METHOD FB_init : BOOL
VAR_INPUT
	bInitRetains : BOOL; // if TRUE, the retain variables are initialized (warm start / cold start)
	bInCopyCode : BOOL;  // if TRUE, the instance afterwards gets moved into the copy code (online change)
	InitialValue : ETcVnCodeDetectionModel;
END_VAR
localData := InitialValue;
AddBaseDatatype(enumBaseDatatype);
ClearReference();

AddLocalEnumeration('TCVN_CDM_DETECT_1_1', ETcVnCodeDetectionModel.TCVN_CDM_DETECT_1_1);
AddLocalEnumeration('TCVN_CDM_DETECT_1_2', ETcVnCodeDetectionModel.TCVN_CDM_DETECT_1_2);
AddLocalEnumeration('TCVN_CDM_DETECT_1_3', ETcVnCodeDetectionModel.TCVN_CDM_DETECT_1_3);
AddLocalEnumeration('TCVN_CDM_DETECT_2_1', ETcVnCodeDetectionModel.TCVN_CDM_DETECT_2_1);
AddLocalEnumeration('TCVN_CDM_DETECT_2_2', ETcVnCodeDetectionModel.TCVN_CDM_DETECT_2_2);
AddLocalEnumeration('TCVN_CDM_DETECT_2_3', ETcVnCodeDetectionModel.TCVN_CDM_DETECT_2_3);
AddLocalEnumeration('TCVN_CDM_DETECT_3_1', ETcVnCodeDetectionModel.TCVN_CDM_DETECT_3_1);
AddLocalEnumeration('TCVN_CDM_DETECT_3_2', ETcVnCodeDetectionModel.TCVN_CDM_DETECT_3_2);
AddLocalEnumeration('TCVN_CDM_DETECT_3_3', ETcVnCodeDetectionModel.TCVN_CDM_DETECT_3_3);
END_METHOD

METHOD PRIVATE AddLocalEnumeration
VAR_INPUT
	Enumeration : T_MAXSTRING;
	Value : ETcVnCodeDetectionModel;
END_VAR
AddEnumeration(Enumeration, Value);
END_METHOD

METHOD IsEnumeratorValueEqual : BOOL
VAR_INPUT
	Enumerator : I_KeyValueForwardEnumerator;
END_VAR
VAR
	storedValue : ETcVnCodeDetectionModel;
END_VAR
IF NOT Enumerator.TryGet(storedValue) THEN
	RETURN;
END_IF

IsEnumeratorValueEqual := storedValue = activeData;
END_METHOD

METHOD PUBLIC Clone : I_Datatype
VAR
    pClone : POINTER TO _ETcVnCodeDetectionModel;
END_VAR
pClone := __NEW(_ETcVnCodeDetectionModel(InitialValue := Value));
Clone := pClone^;
END_METHOD

PROPERTY PUBLIC Identifier : T_MAXSTRING
GET
Identifier := 'ETcVnCodeDetectionModel';
END_GET
END_PROPERTY

METHOD PUBLIC MakeReferenceTo
VAR_INPUT
	ReferenceTarget : REFERENCE TO ETcVnCodeDetectionModel;
END_VAR
activeData REF= ReferenceTarget;
SetBaseDatatypeReference();
END_METHOD

METHOD TryMakeReferenceTo : BOOL
VAR_INPUT
	Target : I_Datatype;
END_VAR
VAR
	pTargetData : POINTER TO ETcVnCodeDetectionModel;
END_VAR
IF NOT IsEquivalentTo(Target) THEN
	RETURN;
END_IF

pTargetData := Target.Address;
activeData REF= pTargetData^;
SetBaseDatatypeReference();
TryMakeReferenceTo := TRUE;
END_METHOD

PROPERTY PUBLIC Value : ETcVnCodeDetectionModel
GET
Value := activeData;
END_GET
SET
activeData := Value;
END_SET
END_PROPERTY

END_FUNCTION_BLOCK

// Datatypes/Enums/_ETcVnCodeType
{attribute 'linkalways'} 
{attribute 'no_explicit_call' := 'This FB is a CLASS and must be accessed using methods or properties'}
{attribute 'enable_dynamic_creation'}
FUNCTION_BLOCK _ETcVnCodeType EXTENDS EnumDatatypeBase
VAR
	localData : ETcVnCodeType;
	activeData : REFERENCE TO ETcVnCodeType;
	enumBaseDatatype : _ULINT(localData);
END_VAR

METHOD PROTECTED SetBaseDatatypeReference
VAR_INPUT
END_VAR
enumBaseDatatype.MakeReferenceTo(activeData);
END_METHOD

PROPERTY PUBLIC Address : PVOID
GET
Address := ADR(activeData);
END_GET
END_PROPERTY

METHOD PUBLIC ClearReference
VAR_INPUT
END_VAR
activeData REF= localData;
SetBaseDatatypeReference();
END_METHOD

PROPERTY PUBLIC Size : UDINT
GET
Size := SIZEOF(activeData);
END_GET
END_PROPERTY

METHOD FB_init : BOOL
VAR_INPUT
	bInitRetains : BOOL; // if TRUE, the retain variables are initialized (warm start / cold start)
	bInCopyCode : BOOL;  // if TRUE, the instance afterwards gets moved into the copy code (online change)
	InitialValue : ETcVnCodeType;
END_VAR
localData := InitialValue;
AddBaseDatatype(enumBaseDatatype);
ClearReference();

AddLocalEnumeration('TCVN_CT_ANY', ETcVnCodeType.TCVN_CT_ANY);
AddLocalEnumeration('TCVN_CT_1D', ETcVnCodeType.TCVN_CT_1D);
AddLocalEnumeration('TCVN_CT_2D', ETcVnCodeType.TCVN_CT_2D);
AddLocalEnumeration('TCVN_CT_QR', ETcVnCodeType.TCVN_CT_QR);
AddLocalEnumeration('TCVN_CT_DATAMATRIX', ETcVnCodeType.TCVN_CT_DATAMATRIX);
AddLocalEnumeration('TCVN_CT_DOTCODE', ETcVnCodeType.TCVN_CT_DOTCODE);
END_METHOD

METHOD PRIVATE AddLocalEnumeration
VAR_INPUT
	Enumeration : T_MAXSTRING;
	Value : ETcVnCodeType;
END_VAR
AddEnumeration(Enumeration, Value);
END_METHOD

METHOD IsEnumeratorValueEqual : BOOL
VAR_INPUT
	Enumerator : I_KeyValueForwardEnumerator;
END_VAR
VAR
	storedValue : ETcVnCodeType;
END_VAR
IF NOT Enumerator.TryGet(storedValue) THEN
	RETURN;
END_IF

IsEnumeratorValueEqual := storedValue = activeData;
END_METHOD

METHOD PUBLIC Clone : I_Datatype
VAR
    pClone : POINTER TO _ETcVnCodeType;
END_VAR
pClone := __NEW(_ETcVnCodeType(InitialValue := Value));
Clone := pClone^;
END_METHOD

PROPERTY PUBLIC Identifier : T_MAXSTRING
GET
Identifier := 'ETcVnCodeType';
END_GET
END_PROPERTY

METHOD PUBLIC MakeReferenceTo
VAR_INPUT
	ReferenceTarget : REFERENCE TO ETcVnCodeType;
END_VAR
activeData REF= ReferenceTarget;
SetBaseDatatypeReference();
END_METHOD

METHOD TryMakeReferenceTo : BOOL
VAR_INPUT
	Target : I_Datatype;
END_VAR
VAR
	pTargetData : POINTER TO ETcVnCodeType;
END_VAR
IF NOT IsEquivalentTo(Target) THEN
	RETURN;
END_IF

pTargetData := Target.Address;
activeData REF= pTargetData^;
SetBaseDatatypeReference();
TryMakeReferenceTo := TRUE;
END_METHOD

PROPERTY PUBLIC Value : ETcVnCodeType
GET
Value := activeData;
END_GET
SET
activeData := Value;
END_SET
END_PROPERTY

END_FUNCTION_BLOCK

// Datatypes/Enums/_ETcVnColorMap
{attribute 'linkalways'} 
{attribute 'no_explicit_call' := 'This FB is a CLASS and must be accessed using methods or properties'}
{attribute 'enable_dynamic_creation'}
FUNCTION_BLOCK _ETcVnColorMap EXTENDS EnumDatatypeBase
VAR
	localData : ETcVnColorMap;
	activeData : REFERENCE TO ETcVnColorMap;
	enumBaseDatatype : _DINT(localData);
END_VAR

METHOD PROTECTED SetBaseDatatypeReference
VAR_INPUT
END_VAR
enumBaseDatatype.MakeReferenceTo(activeData);
END_METHOD

PROPERTY PUBLIC Address : PVOID
GET
Address := ADR(activeData);
END_GET
END_PROPERTY

METHOD PUBLIC ClearReference
VAR_INPUT
END_VAR
activeData REF= localData;
SetBaseDatatypeReference();
END_METHOD

PROPERTY PUBLIC Size : UDINT
GET
Size := SIZEOF(activeData);
END_GET
END_PROPERTY

METHOD FB_init : BOOL
VAR_INPUT
	bInitRetains : BOOL; // if TRUE, the retain variables are initialized (warm start / cold start)
	bInCopyCode : BOOL;  // if TRUE, the instance afterwards gets moved into the copy code (online change)
	InitialValue : ETcVnColorMap;
END_VAR
localData := InitialValue;
AddBaseDatatype(enumBaseDatatype);
ClearReference();

AddLocalEnumeration('TCVN_CM_AUTUMN', ETcVnColorMap.TCVN_CM_AUTUMN);
AddLocalEnumeration('TCVN_CM_BONE', ETcVnColorMap.TCVN_CM_BONE);
AddLocalEnumeration('TCVN_CM_JET', ETcVnColorMap.TCVN_CM_JET);
AddLocalEnumeration('TCVN_CM_WINTER', ETcVnColorMap.TCVN_CM_WINTER);
AddLocalEnumeration('TCVN_CM_RAINBOW', ETcVnColorMap.TCVN_CM_RAINBOW);
AddLocalEnumeration('TCVN_CM_OCEAN', ETcVnColorMap.TCVN_CM_OCEAN);
AddLocalEnumeration('TCVN_CM_SUMMER', ETcVnColorMap.TCVN_CM_SUMMER);
AddLocalEnumeration('TCVN_CM_SPRING', ETcVnColorMap.TCVN_CM_SPRING);
AddLocalEnumeration('TCVN_CM_COOL', ETcVnColorMap.TCVN_CM_COOL);
AddLocalEnumeration('TCVN_CM_HSV', ETcVnColorMap.TCVN_CM_HSV);
AddLocalEnumeration('TCVN_CM_PINK', ETcVnColorMap.TCVN_CM_PINK);
AddLocalEnumeration('TCVN_CM_HOT', ETcVnColorMap.TCVN_CM_HOT);
AddLocalEnumeration('TCVN_CM_PARULA', ETcVnColorMap.TCVN_CM_PARULA);
AddLocalEnumeration('TCVN_CM_MAGMA', ETcVnColorMap.TCVN_CM_MAGMA);
AddLocalEnumeration('TCVN_CM_INFERNO', ETcVnColorMap.TCVN_CM_INFERNO);
AddLocalEnumeration('TCVN_CM_PLASMA', ETcVnColorMap.TCVN_CM_PLASMA);
AddLocalEnumeration('TCVN_CM_VIRIDIS', ETcVnColorMap.TCVN_CM_VIRIDIS);
AddLocalEnumeration('TCVN_CM_CIVIDIS', ETcVnColorMap.TCVN_CM_CIVIDIS);
AddLocalEnumeration('TCVN_CM_TWILIGHT', ETcVnColorMap.TCVN_CM_TWILIGHT);
AddLocalEnumeration('TCVN_CM_TWILIGHT_SHIFTED', ETcVnColorMap.TCVN_CM_TWILIGHT_SHIFTED);
AddLocalEnumeration('TCVN_CM_TURBO', ETcVnColorMap.TCVN_CM_TURBO);
END_METHOD

METHOD PRIVATE AddLocalEnumeration
VAR_INPUT
	Enumeration : T_MAXSTRING;
	Value : ETcVnColorMap;
END_VAR
AddEnumeration(Enumeration, Value);
END_METHOD

METHOD IsEnumeratorValueEqual : BOOL
VAR_INPUT
	Enumerator : I_KeyValueForwardEnumerator;
END_VAR
VAR
	storedValue : ETcVnColorMap;
END_VAR
IF NOT Enumerator.TryGet(storedValue) THEN
	RETURN;
END_IF

IsEnumeratorValueEqual := storedValue = activeData;
END_METHOD

METHOD PUBLIC Clone : I_Datatype
VAR
    pClone : POINTER TO _ETcVnColorMap;
END_VAR
pClone := __NEW(_ETcVnColorMap(InitialValue := Value));
Clone := pClone^;
END_METHOD

PROPERTY PUBLIC Identifier : T_MAXSTRING
GET
Identifier := 'ETcVnColorMap';
END_GET
END_PROPERTY

METHOD PUBLIC MakeReferenceTo
VAR_INPUT
	ReferenceTarget : REFERENCE TO ETcVnCalibrationPatternOrigin;
END_VAR
activeData REF= ReferenceTarget;
SetBaseDatatypeReference();
END_METHOD

METHOD TryMakeReferenceTo : BOOL
VAR_INPUT
	Target : I_Datatype;
END_VAR
VAR
	pTargetData : POINTER TO ETcVnColorMap;
END_VAR
IF NOT IsEquivalentTo(Target) THEN
	RETURN;
END_IF

pTargetData := Target.Address;
activeData REF= pTargetData^;
SetBaseDatatypeReference();
TryMakeReferenceTo := TRUE;
END_METHOD

PROPERTY PUBLIC Value : ETcVnColorMap
GET
Value := activeData;
END_GET
SET
activeData := Value;
END_SET
END_PROPERTY

END_FUNCTION_BLOCK

// Datatypes/Enums/_ETcVnColorMapSize
{attribute 'linkalways'} 
{attribute 'no_explicit_call' := 'This FB is a CLASS and must be accessed using methods or properties'}
{attribute 'enable_dynamic_creation'}
FUNCTION_BLOCK _ETcVnColorMapSize EXTENDS EnumDatatypeBase
VAR
	localData : ETcVnColorMapSize;
	activeData : REFERENCE TO ETcVnColorMapSize;
	enumBaseDatatype : _UDINT(localData);
END_VAR

METHOD PROTECTED SetBaseDatatypeReference
VAR_INPUT
END_VAR
enumBaseDatatype.MakeReferenceTo(activeData);
END_METHOD

PROPERTY PUBLIC Address : PVOID
GET
Address := ADR(activeData);
END_GET
END_PROPERTY

METHOD PUBLIC ClearReference
VAR_INPUT
END_VAR
activeData REF= localData;
SetBaseDatatypeReference();
END_METHOD

PROPERTY PUBLIC Size : UDINT
GET
Size := SIZEOF(activeData);
END_GET
END_PROPERTY

METHOD FB_init : BOOL
VAR_INPUT
	bInitRetains : BOOL; // if TRUE, the retain variables are initialized (warm start / cold start)
	bInCopyCode : BOOL;  // if TRUE, the instance afterwards gets moved into the copy code (online change)
	InitialValue : ETcVnColorMapSize;
END_VAR
localData := InitialValue;
AddBaseDatatype(enumBaseDatatype);
ClearReference();

AddLocalEnumeration('TCVN_CMS_256', ETcVnColorMapSize.TCVN_CMS_256);
AddLocalEnumeration('TCVN_CMS_65536', ETcVnColorMapSize.TCVN_CMS_65536);
END_METHOD

METHOD PRIVATE AddLocalEnumeration
VAR_INPUT
	Enumeration : T_MAXSTRING;
	Value : ETcVnColorMapSize;
END_VAR
AddEnumeration(Enumeration, Value);
END_METHOD

METHOD IsEnumeratorValueEqual : BOOL
VAR_INPUT
	Enumerator : I_KeyValueForwardEnumerator;
END_VAR
VAR
	storedValue : ETcVnColorMapSize;
END_VAR
IF NOT Enumerator.TryGet(storedValue) THEN
	RETURN;
END_IF

IsEnumeratorValueEqual := storedValue = activeData;
END_METHOD

METHOD PUBLIC Clone : I_Datatype
VAR
    pClone : POINTER TO _ETcVnColorMapSize;
END_VAR
pClone := __NEW(_ETcVnColorMapSize(InitialValue := Value));
Clone := pClone^;
END_METHOD

PROPERTY PUBLIC Identifier : T_MAXSTRING
GET
Identifier := 'ETcVnColorMapSize';
END_GET
END_PROPERTY

METHOD PUBLIC MakeReferenceTo
VAR_INPUT
	ReferenceTarget : REFERENCE TO ETcVnColorMapSize;
END_VAR
activeData REF= ReferenceTarget;
SetBaseDatatypeReference();
END_METHOD

METHOD TryMakeReferenceTo : BOOL
VAR_INPUT
	Target : I_Datatype;
END_VAR
VAR
	pTargetData : POINTER TO ETcVnColorMapSize;
END_VAR
IF NOT IsEquivalentTo(Target) THEN
	RETURN;
END_IF

pTargetData := Target.Address;
activeData REF= pTargetData^;
SetBaseDatatypeReference();
TryMakeReferenceTo := TRUE;
END_METHOD

PROPERTY PUBLIC Value : ETcVnColorMapSize
GET
Value := activeData;
END_GET
SET
activeData := Value;
END_SET
END_PROPERTY

END_FUNCTION_BLOCK

// Datatypes/Enums/_ETcVnColorSpaceTransform
{attribute 'linkalways'} 
{attribute 'no_explicit_call' := 'This FB is a CLASS and must be accessed using methods or properties'}
{attribute 'enable_dynamic_creation'}
FUNCTION_BLOCK _ETcVnColorSpaceTransform EXTENDS EnumDatatypeBase
VAR
	localData : ETcVnColorSpaceTransform;
	activeData : REFERENCE TO ETcVnColorSpaceTransform;
	enumBaseDatatype : _DINT(localData);
END_VAR

METHOD PROTECTED SetBaseDatatypeReference
VAR_INPUT
END_VAR
enumBaseDatatype.MakeReferenceTo(activeData);
END_METHOD

PROPERTY PUBLIC Address : PVOID
GET
Address := ADR(activeData);
END_GET
END_PROPERTY

METHOD PUBLIC ClearReference
VAR_INPUT
END_VAR
activeData REF= localData;
SetBaseDatatypeReference();
END_METHOD

PROPERTY PUBLIC Size : UDINT
GET
Size := SIZEOF(activeData);
END_GET
END_PROPERTY

METHOD FB_init : BOOL
VAR_INPUT
	bInitRetains : BOOL; // if TRUE, the retain variables are initialized (warm start / cold start)
	bInCopyCode : BOOL;  // if TRUE, the instance afterwards gets moved into the copy code (online change)
	InitialValue : ETcVnColorSpaceTransform;
END_VAR
localData := InitialValue;
AddBaseDatatype(enumBaseDatatype);
ClearReference();

AddLocalEnumeration('TCVN_CST_BGR_TO_BGRA', ETcVnColorSpaceTransform.TCVN_CST_BGR_TO_BGRA);
AddLocalEnumeration('TCVN_CST_RGB_TO_RGBA', ETcVnColorSpaceTransform.TCVN_CST_RGB_TO_RGBA);
AddLocalEnumeration('TCVN_CST_BGRA_TO_BGR', ETcVnColorSpaceTransform.TCVN_CST_BGRA_TO_BGR);
AddLocalEnumeration('TCVN_CST_RGBA_TO_RGB', ETcVnColorSpaceTransform.TCVN_CST_RGBA_TO_RGB);
AddLocalEnumeration('TCVN_CST_BGR_TO_RGBA', ETcVnColorSpaceTransform.TCVN_CST_BGR_TO_RGBA);
AddLocalEnumeration('TCVN_CST_RGB_TO_BGRA', ETcVnColorSpaceTransform.TCVN_CST_RGB_TO_BGRA);
AddLocalEnumeration('TCVN_CST_BGRA_TO_RGB', ETcVnColorSpaceTransform.TCVN_CST_BGRA_TO_RGB);
AddLocalEnumeration('TCVN_CST_RGBA_TO_BGR', ETcVnColorSpaceTransform.TCVN_CST_RGBA_TO_BGR);
AddLocalEnumeration('TCVN_CST_BGR_TO_RGB', ETcVnColorSpaceTransform.TCVN_CST_BGR_TO_RGB);
AddLocalEnumeration('TCVN_CST_RGB_TO_BGR', ETcVnColorSpaceTransform.TCVN_CST_RGB_TO_BGR);
AddLocalEnumeration('TCVN_CST_BGRA_TO_RGBA', ETcVnColorSpaceTransform.TCVN_CST_BGRA_TO_RGBA);
AddLocalEnumeration('TCVN_CST_RGBA_TO_BGRA', ETcVnColorSpaceTransform.TCVN_CST_RGBA_TO_BGRA);
AddLocalEnumeration('TCVN_CST_BGR_TO_GRAY', ETcVnColorSpaceTransform.TCVN_CST_BGR_TO_GRAY);
AddLocalEnumeration('TCVN_CST_RGB_TO_GRAY', ETcVnColorSpaceTransform.TCVN_CST_RGB_TO_GRAY);
AddLocalEnumeration('TCVN_CST_GRAY_TO_BGR', ETcVnColorSpaceTransform.TCVN_CST_GRAY_TO_BGR);
AddLocalEnumeration('TCVN_CST_GRAY_TO_RGB', ETcVnColorSpaceTransform.TCVN_CST_GRAY_TO_RGB);
AddLocalEnumeration('TCVN_CST_GRAY_TO_BGRA', ETcVnColorSpaceTransform.TCVN_CST_GRAY_TO_BGRA);
AddLocalEnumeration('TCVN_CST_GRAY_TO_RGBA', ETcVnColorSpaceTransform.TCVN_CST_GRAY_TO_RGBA);
AddLocalEnumeration('TCVN_CST_BGRA_TO_GRAY', ETcVnColorSpaceTransform.TCVN_CST_BGRA_TO_GRAY);
AddLocalEnumeration('TCVN_CST_RGBA_TO_GRAY', ETcVnColorSpaceTransform.TCVN_CST_RGBA_TO_GRAY);
AddLocalEnumeration('TCVN_CST_RGB_TO_BGR_565', ETcVnColorSpaceTransform.TCVN_CST_RGB_TO_BGR_565);
AddLocalEnumeration('TCVN_CST_BGR_TO_BGR_565', ETcVnColorSpaceTransform.TCVN_CST_BGR_TO_BGR_565);
AddLocalEnumeration('TCVN_CST_BGR_565_TO_RGB', ETcVnColorSpaceTransform.TCVN_CST_BGR_565_TO_RGB);
AddLocalEnumeration('TCVN_CST_BGR_565_TO_BGR', ETcVnColorSpaceTransform.TCVN_CST_BGR_565_TO_BGR);
AddLocalEnumeration('TCVN_CST_RGBA_TO_BGR_565', ETcVnColorSpaceTransform.TCVN_CST_RGBA_TO_BGR_565);
AddLocalEnumeration('TCVN_CST_BGRA_TO_BGR_565', ETcVnColorSpaceTransform.TCVN_CST_BGRA_TO_BGR_565);
AddLocalEnumeration('TCVN_CST_BGR_565_TO_RGBA', ETcVnColorSpaceTransform.TCVN_CST_BGR_565_TO_RGBA);
AddLocalEnumeration('TCVN_CST_BGR_565_TO_BGRA', ETcVnColorSpaceTransform.TCVN_CST_BGR_565_TO_BGRA);
AddLocalEnumeration('TCVN_CST_GRAY_TO_BGR_565', ETcVnColorSpaceTransform.TCVN_CST_GRAY_TO_BGR_565);
AddLocalEnumeration('TCVN_CST_BGR_565_TO_GRAY', ETcVnColorSpaceTransform.TCVN_CST_BGR_565_TO_GRAY);
AddLocalEnumeration('TCVN_CST_RGB_TO_BGR_555', ETcVnColorSpaceTransform.TCVN_CST_RGB_TO_BGR_555);
AddLocalEnumeration('TCVN_CST_BGR_TO_BGR_555', ETcVnColorSpaceTransform.TCVN_CST_BGR_TO_BGR_555);
AddLocalEnumeration('TCVN_CST_BGR_555_TO_RGB', ETcVnColorSpaceTransform.TCVN_CST_BGR_555_TO_RGB);
AddLocalEnumeration('TCVN_CST_BGR_555_TO_BGR', ETcVnColorSpaceTransform.TCVN_CST_BGR_555_TO_BGR);
AddLocalEnumeration('TCVN_CST_RGBA_TO_BGR_555', ETcVnColorSpaceTransform.TCVN_CST_RGBA_TO_BGR_555);
AddLocalEnumeration('TCVN_CST_BGRA_TO_BGR_555', ETcVnColorSpaceTransform.TCVN_CST_BGRA_TO_BGR_555);
AddLocalEnumeration('TCVN_CST_BGR_555_TO_RGBA', ETcVnColorSpaceTransform.TCVN_CST_BGR_555_TO_RGBA);
AddLocalEnumeration('TCVN_CST_BGR_555_TO_BGRA', ETcVnColorSpaceTransform.TCVN_CST_BGR_555_TO_BGRA);
AddLocalEnumeration('TCVN_CST_GRAY_TO_BGR_555', ETcVnColorSpaceTransform.TCVN_CST_GRAY_TO_BGR_555);
AddLocalEnumeration('TCVN_CST_BGR_555_TO_GRAY', ETcVnColorSpaceTransform.TCVN_CST_BGR_555_TO_GRAY);
AddLocalEnumeration('TCVN_CST_BGR_TO_XYZ', ETcVnColorSpaceTransform.TCVN_CST_BGR_TO_XYZ);
AddLocalEnumeration('TCVN_CST_RGB_TO_XYZ', ETcVnColorSpaceTransform.TCVN_CST_RGB_TO_XYZ);
AddLocalEnumeration('TCVN_CST_XYZ_TO_BGR', ETcVnColorSpaceTransform.TCVN_CST_XYZ_TO_BGR);
AddLocalEnumeration('TCVN_CST_XYZ_TO_RGB', ETcVnColorSpaceTransform.TCVN_CST_XYZ_TO_RGB);
AddLocalEnumeration('TCVN_CST_BGR_TO_YCRCB', ETcVnColorSpaceTransform.TCVN_CST_BGR_TO_YCRCB);
AddLocalEnumeration('TCVN_CST_RGB_TO_YCRCB', ETcVnColorSpaceTransform.TCVN_CST_RGB_TO_YCRCB);
AddLocalEnumeration('TCVN_CST_YCRCB_TO_BGR', ETcVnColorSpaceTransform.TCVN_CST_YCRCB_TO_BGR);
AddLocalEnumeration('TCVN_CST_YCRCB_TO_RGB', ETcVnColorSpaceTransform.TCVN_CST_YCRCB_TO_RGB);
AddLocalEnumeration('TCVN_CST_BGR_TO_HSV', ETcVnColorSpaceTransform.TCVN_CST_BGR_TO_HSV);
AddLocalEnumeration('TCVN_CST_RGB_TO_HSV', ETcVnColorSpaceTransform.TCVN_CST_RGB_TO_HSV);
AddLocalEnumeration('TCVN_CST_BGR_TO_LAB', ETcVnColorSpaceTransform.TCVN_CST_BGR_TO_LAB);
AddLocalEnumeration('TCVN_CST_RGB_TO_LAB', ETcVnColorSpaceTransform.TCVN_CST_RGB_TO_LAB);
AddLocalEnumeration('TCVN_CST_BAYER_RG_TO_BGR', ETcVnColorSpaceTransform.TCVN_CST_BAYER_RG_TO_BGR);
AddLocalEnumeration('TCVN_CST_BAYER_BG_TO_RGB', ETcVnColorSpaceTransform.TCVN_CST_BAYER_BG_TO_RGB);
AddLocalEnumeration('TCVN_CST_BAYER_GR_TO_BGR', ETcVnColorSpaceTransform.TCVN_CST_BAYER_GR_TO_BGR);
AddLocalEnumeration('TCVN_CST_BAYER_GB_TO_RGB', ETcVnColorSpaceTransform.TCVN_CST_BAYER_GB_TO_RGB);
AddLocalEnumeration('TCVN_CST_BAYER_BG_TO_BGR', ETcVnColorSpaceTransform.TCVN_CST_BAYER_BG_TO_BGR);
AddLocalEnumeration('TCVN_CST_BAYER_RG_TO_RGB', ETcVnColorSpaceTransform.TCVN_CST_BAYER_RG_TO_RGB);
AddLocalEnumeration('TCVN_CST_BAYER_GB_TO_BGR', ETcVnColorSpaceTransform.TCVN_CST_BAYER_GB_TO_BGR);
AddLocalEnumeration('TCVN_CST_BAYER_GR_TO_RGB', ETcVnColorSpaceTransform.TCVN_CST_BAYER_GR_TO_RGB);
AddLocalEnumeration('TCVN_CST_BGR_TO_LUV', ETcVnColorSpaceTransform.TCVN_CST_BGR_TO_LUV);
AddLocalEnumeration('TCVN_CST_RGB_TO_LUV', ETcVnColorSpaceTransform.TCVN_CST_RGB_TO_LUV);
AddLocalEnumeration('TCVN_CST_BGR_TO_HLS', ETcVnColorSpaceTransform.TCVN_CST_BGR_TO_HLS);
AddLocalEnumeration('TCVN_CST_RGB_TO_HLS', ETcVnColorSpaceTransform.TCVN_CST_RGB_TO_HLS);
AddLocalEnumeration('TCVN_CST_HSV_TO_BGR', ETcVnColorSpaceTransform.TCVN_CST_HSV_TO_BGR);
AddLocalEnumeration('TCVN_CST_HSV_TO_RGB', ETcVnColorSpaceTransform.TCVN_CST_HSV_TO_RGB);
AddLocalEnumeration('TCVN_CST_LAB_TO_BGR', ETcVnColorSpaceTransform.TCVN_CST_LAB_TO_BGR);
AddLocalEnumeration('TCVN_CST_LAB_TO_RGB', ETcVnColorSpaceTransform.TCVN_CST_LAB_TO_RGB);
AddLocalEnumeration('TCVN_CST_LUV_TO_BGR', ETcVnColorSpaceTransform.TCVN_CST_LUV_TO_BGR);
AddLocalEnumeration('TCVN_CST_LUV_TO_RGB', ETcVnColorSpaceTransform.TCVN_CST_LUV_TO_RGB);
AddLocalEnumeration('TCVN_CST_HLS_TO_BGR', ETcVnColorSpaceTransform.TCVN_CST_HLS_TO_BGR);
AddLocalEnumeration('TCVN_CST_HLS_TO_RGB', ETcVnColorSpaceTransform.TCVN_CST_HLS_TO_RGB);
AddLocalEnumeration('TCVN_CST_BAYER_RG_TO_BGR_VNG', ETcVnColorSpaceTransform.TCVN_CST_BAYER_RG_TO_BGR_VNG);
AddLocalEnumeration('TCVN_CST_BAYER_GR_TO_BGR_VNG', ETcVnColorSpaceTransform.TCVN_CST_BAYER_GR_TO_BGR_VNG);
AddLocalEnumeration('TCVN_CST_BAYER_BG_TO_BGR_VNG', ETcVnColorSpaceTransform.TCVN_CST_BAYER_BG_TO_BGR_VNG);
AddLocalEnumeration('TCVN_CST_BAYER_GB_TO_BGR_VNG', ETcVnColorSpaceTransform.TCVN_CST_BAYER_GB_TO_BGR_VNG);
AddLocalEnumeration('TCVN_CST_BAYER_RG_TO_RGB_VNG', ETcVnColorSpaceTransform.TCVN_CST_BAYER_RG_TO_RGB_VNG);
AddLocalEnumeration('TCVN_CST_BAYER_GR_TO_RGB_VNG', ETcVnColorSpaceTransform.TCVN_CST_BAYER_GR_TO_RGB_VNG);
AddLocalEnumeration('TCVN_CST_BAYER_BG_TO_RGB_VNG', ETcVnColorSpaceTransform.TCVN_CST_BAYER_BG_TO_RGB_VNG);
AddLocalEnumeration('TCVN_CST_BAYER_GB_TO_RGB_VNG', ETcVnColorSpaceTransform.TCVN_CST_BAYER_GB_TO_RGB_VNG);
AddLocalEnumeration('TCVN_CST_BGR_TO_HSV_FULL', ETcVnColorSpaceTransform.TCVN_CST_BGR_TO_HSV_FULL);
AddLocalEnumeration('TCVN_CST_RGB_TO_HSV_FULL', ETcVnColorSpaceTransform.TCVN_CST_RGB_TO_HSV_FULL);
AddLocalEnumeration('TCVN_CST_BGR_TO_HLS_FULL', ETcVnColorSpaceTransform.TCVN_CST_BGR_TO_HLS_FULL);
AddLocalEnumeration('TCVN_CST_RGB_TO_HLS_FULL', ETcVnColorSpaceTransform.TCVN_CST_RGB_TO_HLS_FULL);
AddLocalEnumeration('TCVN_CST_HSV_TO_BGR_FULL', ETcVnColorSpaceTransform.TCVN_CST_HSV_TO_BGR_FULL);
AddLocalEnumeration('TCVN_CST_HSV_TO_RGB_FULL', ETcVnColorSpaceTransform.TCVN_CST_HSV_TO_RGB_FULL);
AddLocalEnumeration('TCVN_CST_HLS_TO_BGR_FULL', ETcVnColorSpaceTransform.TCVN_CST_HLS_TO_BGR_FULL);
AddLocalEnumeration('TCVN_CST_HLS_TO_RGB_FULL', ETcVnColorSpaceTransform.TCVN_CST_HLS_TO_RGB_FULL);
AddLocalEnumeration('TCVN_CST_LBGR_TO_LAB', ETcVnColorSpaceTransform.TCVN_CST_LBGR_TO_LAB);
AddLocalEnumeration('TCVN_CST_LRGB_TO_LAB', ETcVnColorSpaceTransform.TCVN_CST_LRGB_TO_LAB);
AddLocalEnumeration('TCVN_CST_LBGR_TO_LUV', ETcVnColorSpaceTransform.TCVN_CST_LBGR_TO_LUV);
AddLocalEnumeration('TCVN_CST_LRGB_TO_LUV', ETcVnColorSpaceTransform.TCVN_CST_LRGB_TO_LUV);
AddLocalEnumeration('TCVN_CST_LAB_TO_LBGR', ETcVnColorSpaceTransform.TCVN_CST_LAB_TO_LBGR);
AddLocalEnumeration('TCVN_CST_LAB_TO_LRGB', ETcVnColorSpaceTransform.TCVN_CST_LAB_TO_LRGB);
AddLocalEnumeration('TCVN_CST_LUV_TO_LBGR', ETcVnColorSpaceTransform.TCVN_CST_LUV_TO_LBGR);
AddLocalEnumeration('TCVN_CST_LUV_TO_LRGB', ETcVnColorSpaceTransform.TCVN_CST_LUV_TO_LRGB);
AddLocalEnumeration('TCVN_CST_BGR_TO_YUV', ETcVnColorSpaceTransform.TCVN_CST_BGR_TO_YUV);
AddLocalEnumeration('TCVN_CST_RGB_TO_YUV', ETcVnColorSpaceTransform.TCVN_CST_RGB_TO_YUV);
AddLocalEnumeration('TCVN_CST_YUV_TO_BGR', ETcVnColorSpaceTransform.TCVN_CST_YUV_TO_BGR);
AddLocalEnumeration('TCVN_CST_YUV_TO_RGB', ETcVnColorSpaceTransform.TCVN_CST_YUV_TO_RGB);
AddLocalEnumeration('TCVN_CST_BAYER_RG_TO_GRAY', ETcVnColorSpaceTransform.TCVN_CST_BAYER_RG_TO_GRAY);
AddLocalEnumeration('TCVN_CST_BAYER_GR_TO_GRAY', ETcVnColorSpaceTransform.TCVN_CST_BAYER_GR_TO_GRAY);
AddLocalEnumeration('TCVN_CST_BAYER_BG_TO_GRAY', ETcVnColorSpaceTransform.TCVN_CST_BAYER_BG_TO_GRAY);
AddLocalEnumeration('TCVN_CST_BAYER_GB_TO_GRAY', ETcVnColorSpaceTransform.TCVN_CST_BAYER_GB_TO_GRAY);
AddLocalEnumeration('TCVN_CST_YUV_420_NV12_TO_RGB', ETcVnColorSpaceTransform.TCVN_CST_YUV_420_NV12_TO_RGB);
AddLocalEnumeration('TCVN_CST_YUV_420_NV12_TO_BGR', ETcVnColorSpaceTransform.TCVN_CST_YUV_420_NV12_TO_BGR);
AddLocalEnumeration('TCVN_CST_YUV_420_NV21_TO_RGB', ETcVnColorSpaceTransform.TCVN_CST_YUV_420_NV21_TO_RGB);
AddLocalEnumeration('TCVN_CST_YUV_420_NV21_TO_BGR', ETcVnColorSpaceTransform.TCVN_CST_YUV_420_NV21_TO_BGR);
AddLocalEnumeration('TCVN_CST_YUV_420_SP_TO_RGB', ETcVnColorSpaceTransform.TCVN_CST_YUV_420_SP_TO_RGB);
AddLocalEnumeration('TCVN_CST_YUV_420_SP_TO_BGR', ETcVnColorSpaceTransform.TCVN_CST_YUV_420_SP_TO_BGR);
AddLocalEnumeration('TCVN_CST_YUV_420_NV12_TO_RGBA', ETcVnColorSpaceTransform.TCVN_CST_YUV_420_NV12_TO_RGBA);
AddLocalEnumeration('TCVN_CST_YUV_420_NV12_TO_BGRA', ETcVnColorSpaceTransform.TCVN_CST_YUV_420_NV12_TO_BGRA);
AddLocalEnumeration('TCVN_CST_YUV_420_NV21_TO_RGBA', ETcVnColorSpaceTransform.TCVN_CST_YUV_420_NV21_TO_RGBA);
AddLocalEnumeration('TCVN_CST_YUV_420_NV21_TO_BGRA', ETcVnColorSpaceTransform.TCVN_CST_YUV_420_NV21_TO_BGRA);
AddLocalEnumeration('TCVN_CST_YUV_420_SP_TO_RGBA', ETcVnColorSpaceTransform.TCVN_CST_YUV_420_SP_TO_RGBA);
AddLocalEnumeration('TCVN_CST_YUV_420_SP_TO_BGRA', ETcVnColorSpaceTransform.TCVN_CST_YUV_420_SP_TO_BGRA);
AddLocalEnumeration('TCVN_CST_YUV_420_YV12_TO_RGB', ETcVnColorSpaceTransform.TCVN_CST_YUV_420_YV12_TO_RGB);
AddLocalEnumeration('TCVN_CST_YUV_420_YV12_TO_BGR', ETcVnColorSpaceTransform.TCVN_CST_YUV_420_YV12_TO_BGR);
AddLocalEnumeration('TCVN_CST_YUV_420_IYUV_TO_RGB', ETcVnColorSpaceTransform.TCVN_CST_YUV_420_IYUV_TO_RGB);
AddLocalEnumeration('TCVN_CST_YUV_420_IYUV_TO_BGR', ETcVnColorSpaceTransform.TCVN_CST_YUV_420_IYUV_TO_BGR);
AddLocalEnumeration('TCVN_CST_YUV_420_I420_TO_RGB', ETcVnColorSpaceTransform.TCVN_CST_YUV_420_I420_TO_RGB);
AddLocalEnumeration('TCVN_CST_YUV_420_I420_TO_BGR', ETcVnColorSpaceTransform.TCVN_CST_YUV_420_I420_TO_BGR);
AddLocalEnumeration('TCVN_CST_YUV_420_P_TO_RGB', ETcVnColorSpaceTransform.TCVN_CST_YUV_420_P_TO_RGB);
AddLocalEnumeration('TCVN_CST_YUV_420_P_TO_BGR', ETcVnColorSpaceTransform.TCVN_CST_YUV_420_P_TO_BGR);
AddLocalEnumeration('TCVN_CST_YUV_420_YV12_TO_RGBA', ETcVnColorSpaceTransform.TCVN_CST_YUV_420_YV12_TO_RGBA);
AddLocalEnumeration('TCVN_CST_YUV_420_YV12_TO_BGRA', ETcVnColorSpaceTransform.TCVN_CST_YUV_420_YV12_TO_BGRA);
AddLocalEnumeration('TCVN_CST_YUV_420_IYUV_TO_RGBA', ETcVnColorSpaceTransform.TCVN_CST_YUV_420_IYUV_TO_RGBA);
AddLocalEnumeration('TCVN_CST_YUV_420_IYUV_TO_BGRA', ETcVnColorSpaceTransform.TCVN_CST_YUV_420_IYUV_TO_BGRA);
AddLocalEnumeration('TCVN_CST_YUV_420_I420_TO_RGBA', ETcVnColorSpaceTransform.TCVN_CST_YUV_420_I420_TO_RGBA);
AddLocalEnumeration('TCVN_CST_YUV_420_I420_TO_BGRA', ETcVnColorSpaceTransform.TCVN_CST_YUV_420_I420_TO_BGRA);
AddLocalEnumeration('TCVN_CST_YUV_420_P_TO_RGBA', ETcVnColorSpaceTransform.TCVN_CST_YUV_420_P_TO_RGBA);
AddLocalEnumeration('TCVN_CST_YUV_420_P_TO_BGRA', ETcVnColorSpaceTransform.TCVN_CST_YUV_420_P_TO_BGRA);
AddLocalEnumeration('TCVN_CST_YUV_420_TO_GRAY', ETcVnColorSpaceTransform.TCVN_CST_YUV_420_TO_GRAY);
AddLocalEnumeration('TCVN_CST_YUV_420_NV21_TO_GRAY', ETcVnColorSpaceTransform.TCVN_CST_YUV_420_NV21_TO_GRAY);
AddLocalEnumeration('TCVN_CST_YUV_420_NV12_TO_GRAY', ETcVnColorSpaceTransform.TCVN_CST_YUV_420_NV12_TO_GRAY);
AddLocalEnumeration('TCVN_CST_YUV_420_YV12_TO_GRAY', ETcVnColorSpaceTransform.TCVN_CST_YUV_420_YV12_TO_GRAY);
AddLocalEnumeration('TCVN_CST_YUV_420_IYUV_TO_GRAY', ETcVnColorSpaceTransform.TCVN_CST_YUV_420_IYUV_TO_GRAY);
AddLocalEnumeration('TCVN_CST_YUV_420_I420_TO_GRAY', ETcVnColorSpaceTransform.TCVN_CST_YUV_420_I420_TO_GRAY);
AddLocalEnumeration('TCVN_CST_YUV_420_SP_TO_GRAY', ETcVnColorSpaceTransform.TCVN_CST_YUV_420_SP_TO_GRAY);
AddLocalEnumeration('TCVN_CST_YUV_420_P_TO_GRAY', ETcVnColorSpaceTransform.TCVN_CST_YUV_420_P_TO_GRAY);
AddLocalEnumeration('TCVN_CST_YUV_422_UYVY_TO_RGB', ETcVnColorSpaceTransform.TCVN_CST_YUV_422_UYVY_TO_RGB);
AddLocalEnumeration('TCVN_CST_YUV_422_UYVY_TO_BGR', ETcVnColorSpaceTransform.TCVN_CST_YUV_422_UYVY_TO_BGR);
AddLocalEnumeration('TCVN_CST_YUV_422_Y422_TO_RGB', ETcVnColorSpaceTransform.TCVN_CST_YUV_422_Y422_TO_RGB);
AddLocalEnumeration('TCVN_CST_YUV_422_Y422_TO_BGR', ETcVnColorSpaceTransform.TCVN_CST_YUV_422_Y422_TO_BGR);
AddLocalEnumeration('TCVN_CST_YUV_422_UYNV_TO_RGB', ETcVnColorSpaceTransform.TCVN_CST_YUV_422_UYNV_TO_RGB);
AddLocalEnumeration('TCVN_CST_YUV_422_UYNV_TO_BGR', ETcVnColorSpaceTransform.TCVN_CST_YUV_422_UYNV_TO_BGR);
AddLocalEnumeration('TCVN_CST_YUV_422_UYVY_TO_RGBA', ETcVnColorSpaceTransform.TCVN_CST_YUV_422_UYVY_TO_RGBA);
AddLocalEnumeration('TCVN_CST_YUV_422_UYVY_TO_BGRA', ETcVnColorSpaceTransform.TCVN_CST_YUV_422_UYVY_TO_BGRA);
AddLocalEnumeration('TCVN_CST_YUV_422_Y422_TO_RGBA', ETcVnColorSpaceTransform.TCVN_CST_YUV_422_Y422_TO_RGBA);
AddLocalEnumeration('TCVN_CST_YUV_422_Y422_TO_BGRA', ETcVnColorSpaceTransform.TCVN_CST_YUV_422_Y422_TO_BGRA);
AddLocalEnumeration('TCVN_CST_YUV_422_UYNV_TO_RGBA', ETcVnColorSpaceTransform.TCVN_CST_YUV_422_UYNV_TO_RGBA);
AddLocalEnumeration('TCVN_CST_YUV_422_UYNV_TO_BGRA', ETcVnColorSpaceTransform.TCVN_CST_YUV_422_UYNV_TO_BGRA);
AddLocalEnumeration('TCVN_CST_YUV_422_YUY2_TO_RGB', ETcVnColorSpaceTransform.TCVN_CST_YUV_422_YUY2_TO_RGB);
AddLocalEnumeration('TCVN_CST_YUV_422_YUY2_TO_BGR', ETcVnColorSpaceTransform.TCVN_CST_YUV_422_YUY2_TO_BGR);
AddLocalEnumeration('TCVN_CST_YUV_422_YVYU_TO_RGB', ETcVnColorSpaceTransform.TCVN_CST_YUV_422_YVYU_TO_RGB);
AddLocalEnumeration('TCVN_CST_YUV_422_YVYU_TO_BGR', ETcVnColorSpaceTransform.TCVN_CST_YUV_422_YVYU_TO_BGR);
AddLocalEnumeration('TCVN_CST_YUV_422_YUYV_TO_RGB', ETcVnColorSpaceTransform.TCVN_CST_YUV_422_YUYV_TO_RGB);
AddLocalEnumeration('TCVN_CST_YUV_422_YUYV_TO_BGR', ETcVnColorSpaceTransform.TCVN_CST_YUV_422_YUYV_TO_BGR);
AddLocalEnumeration('TCVN_CST_YUV_422_YUNV_TO_RGB', ETcVnColorSpaceTransform.TCVN_CST_YUV_422_YUNV_TO_RGB);
AddLocalEnumeration('TCVN_CST_YUV_422_YUNV_TO_BGR', ETcVnColorSpaceTransform.TCVN_CST_YUV_422_YUNV_TO_BGR);
AddLocalEnumeration('TCVN_CST_YUV_422_YUY2_TO_RGBA', ETcVnColorSpaceTransform.TCVN_CST_YUV_422_YUY2_TO_RGBA);
AddLocalEnumeration('TCVN_CST_YUV_422_YUY2_TO_BGRA', ETcVnColorSpaceTransform.TCVN_CST_YUV_422_YUY2_TO_BGRA);
AddLocalEnumeration('TCVN_CST_YUV_422_YVYU_TO_RGBA', ETcVnColorSpaceTransform.TCVN_CST_YUV_422_YVYU_TO_RGBA);
AddLocalEnumeration('TCVN_CST_YUV_422_YVYU_TO_BGRA', ETcVnColorSpaceTransform.TCVN_CST_YUV_422_YVYU_TO_BGRA);
AddLocalEnumeration('TCVN_CST_YUV_422_YUYV_TO_RGBA', ETcVnColorSpaceTransform.TCVN_CST_YUV_422_YUYV_TO_RGBA);
AddLocalEnumeration('TCVN_CST_YUV_422_YUYV_TO_BGRA', ETcVnColorSpaceTransform.TCVN_CST_YUV_422_YUYV_TO_BGRA);
AddLocalEnumeration('TCVN_CST_YUV_422_YUNV_TO_RGBA', ETcVnColorSpaceTransform.TCVN_CST_YUV_422_YUNV_TO_RGBA);
AddLocalEnumeration('TCVN_CST_YUV_422_YUNV_TO_BGRA', ETcVnColorSpaceTransform.TCVN_CST_YUV_422_YUNV_TO_BGRA);
AddLocalEnumeration('TCVN_CST_YUV_422_UYVY_TO_GRAY', ETcVnColorSpaceTransform.TCVN_CST_YUV_422_UYVY_TO_GRAY);
AddLocalEnumeration('TCVN_CST_YUV_422_YUY2_TO_GRAY', ETcVnColorSpaceTransform.TCVN_CST_YUV_422_YUY2_TO_GRAY);
AddLocalEnumeration('TCVN_CST_YUV_422_Y422_TO_GRAY', ETcVnColorSpaceTransform.TCVN_CST_YUV_422_Y422_TO_GRAY);
AddLocalEnumeration('TCVN_CST_YUV_422_UYNV_TO_GRAY', ETcVnColorSpaceTransform.TCVN_CST_YUV_422_UYNV_TO_GRAY);
AddLocalEnumeration('TCVN_CST_YUV_422_YVYU_TO_GRAY', ETcVnColorSpaceTransform.TCVN_CST_YUV_422_YVYU_TO_GRAY);
AddLocalEnumeration('TCVN_CST_YUV_422_YUYV_TO_GRAY', ETcVnColorSpaceTransform.TCVN_CST_YUV_422_YUYV_TO_GRAY);
AddLocalEnumeration('TCVN_CST_YUV_422_YUNV_TO_GRAY', ETcVnColorSpaceTransform.TCVN_CST_YUV_422_YUNV_TO_GRAY);
AddLocalEnumeration('TCVN_CST_RGBA_TO_PREMULTIPLICATED_RGBA', ETcVnColorSpaceTransform.TCVN_CST_RGBA_TO_PREMULTIPLICATED_RGBA);
AddLocalEnumeration('TCVN_CST_PREMULTIPLICATED_RGBA_TO_RGBA', ETcVnColorSpaceTransform.TCVN_CST_PREMULTIPLICATED_RGBA_TO_RGBA);
AddLocalEnumeration('TCVN_CST_RGB_TO_YUV_420_I420', ETcVnColorSpaceTransform.TCVN_CST_RGB_TO_YUV_420_I420);
AddLocalEnumeration('TCVN_CST_BGR_TO_YUV_420_I420', ETcVnColorSpaceTransform.TCVN_CST_BGR_TO_YUV_420_I420);
AddLocalEnumeration('TCVN_CST_RGB_TO_YUV_420_IYUV', ETcVnColorSpaceTransform.TCVN_CST_RGB_TO_YUV_420_IYUV);
AddLocalEnumeration('TCVN_CST_BGR_TO_YUV_420_IYUV', ETcVnColorSpaceTransform.TCVN_CST_BGR_TO_YUV_420_IYUV);
AddLocalEnumeration('TCVN_CST_RGBA_TO_YUV_420_I420', ETcVnColorSpaceTransform.TCVN_CST_RGBA_TO_YUV_420_I420);
AddLocalEnumeration('TCVN_CST_BGRA_TO_YUV_420_I420', ETcVnColorSpaceTransform.TCVN_CST_BGRA_TO_YUV_420_I420);
AddLocalEnumeration('TCVN_CST_RGBA_TO_YUV_420_IYUV', ETcVnColorSpaceTransform.TCVN_CST_RGBA_TO_YUV_420_IYUV);
AddLocalEnumeration('TCVN_CST_BGRA_TO_YUV_420_IYUV', ETcVnColorSpaceTransform.TCVN_CST_BGRA_TO_YUV_420_IYUV);
AddLocalEnumeration('TCVN_CST_RGB_TO_YUV_420_YV12', ETcVnColorSpaceTransform.TCVN_CST_RGB_TO_YUV_420_YV12);
AddLocalEnumeration('TCVN_CST_BGR_TO_YUV_420_YV12', ETcVnColorSpaceTransform.TCVN_CST_BGR_TO_YUV_420_YV12);
AddLocalEnumeration('TCVN_CST_RGBA_TO_YUV_420_YV12', ETcVnColorSpaceTransform.TCVN_CST_RGBA_TO_YUV_420_YV12);
AddLocalEnumeration('TCVN_CST_BGRA_TO_YUV_420_YV12', ETcVnColorSpaceTransform.TCVN_CST_BGRA_TO_YUV_420_YV12);
AddLocalEnumeration('TCVN_CST_BAYER_RG_TO_BGR_EA', ETcVnColorSpaceTransform.TCVN_CST_BAYER_RG_TO_BGR_EA);
AddLocalEnumeration('TCVN_CST_BAYER_GR_TO_BGR_EA', ETcVnColorSpaceTransform.TCVN_CST_BAYER_GR_TO_BGR_EA);
AddLocalEnumeration('TCVN_CST_BAYER_BG_TO_BGR_EA', ETcVnColorSpaceTransform.TCVN_CST_BAYER_BG_TO_BGR_EA);
AddLocalEnumeration('TCVN_CST_BAYER_GB_TO_BGR_EA', ETcVnColorSpaceTransform.TCVN_CST_BAYER_GB_TO_BGR_EA);
AddLocalEnumeration('TCVN_CST_BAYER_RG_TO_RGB_EA', ETcVnColorSpaceTransform.TCVN_CST_BAYER_RG_TO_RGB_EA);
AddLocalEnumeration('TCVN_CST_BAYER_GR_TO_RGB_EA', ETcVnColorSpaceTransform.TCVN_CST_BAYER_GR_TO_RGB_EA);
AddLocalEnumeration('TCVN_CST_BAYER_BG_TO_RGB_EA', ETcVnColorSpaceTransform.TCVN_CST_BAYER_BG_TO_RGB_EA);
AddLocalEnumeration('TCVN_CST_BAYER_GB_TO_RGB_EA', ETcVnColorSpaceTransform.TCVN_CST_BAYER_GB_TO_RGB_EA);
AddLocalEnumeration('TCVN_CST_BAYER_RG_TO_BGRA', ETcVnColorSpaceTransform.TCVN_CST_BAYER_RG_TO_BGRA);
AddLocalEnumeration('TCVN_CST_BAYER_GR_TO_BGRA', ETcVnColorSpaceTransform.TCVN_CST_BAYER_GR_TO_BGRA);
AddLocalEnumeration('TCVN_CST_BAYER_BG_TO_BGRA', ETcVnColorSpaceTransform.TCVN_CST_BAYER_BG_TO_BGRA);
AddLocalEnumeration('TCVN_CST_BAYER_GB_TO_BGRA', ETcVnColorSpaceTransform.TCVN_CST_BAYER_GB_TO_BGRA);
AddLocalEnumeration('TCVN_CST_BAYER_RG_TO_RGBA', ETcVnColorSpaceTransform.TCVN_CST_BAYER_RG_TO_RGBA);
AddLocalEnumeration('TCVN_CST_BAYER_GR_TO_RGBA', ETcVnColorSpaceTransform.TCVN_CST_BAYER_GR_TO_RGBA);
AddLocalEnumeration('TCVN_CST_BAYER_BG_TO_RGBA', ETcVnColorSpaceTransform.TCVN_CST_BAYER_BG_TO_RGBA);
AddLocalEnumeration('TCVN_CST_BAYER_GB_TO_RGBA', ETcVnColorSpaceTransform.TCVN_CST_BAYER_GB_TO_RGBA);
AddLocalEnumeration('TCVN_CST_MAX', ETcVnColorSpaceTransform.TCVN_CST_MAX);
AddLocalEnumeration('TCVN_CST_RGB_TO_YUV_422_UYVY', ETcVnColorSpaceTransform.TCVN_CST_RGB_TO_YUV_422_UYVY);
AddLocalEnumeration('TCVN_CST_BGR_TO_YUV_422_UYVY', ETcVnColorSpaceTransform.TCVN_CST_BGR_TO_YUV_422_UYVY);
AddLocalEnumeration('TCVN_CST_RGB_TO_YUV_422_Y422', ETcVnColorSpaceTransform.TCVN_CST_RGB_TO_YUV_422_Y422);
AddLocalEnumeration('TCVN_CST_BGR_TO_YUV_422_Y422', ETcVnColorSpaceTransform.TCVN_CST_BGR_TO_YUV_422_Y422);
AddLocalEnumeration('TCVN_CST_RGB_TO_YUV_422_UYNV', ETcVnColorSpaceTransform.TCVN_CST_RGB_TO_YUV_422_UYNV);
AddLocalEnumeration('TCVN_CST_BGR_TO_YUV_422_UYNV', ETcVnColorSpaceTransform.TCVN_CST_BGR_TO_YUV_422_UYNV);
AddLocalEnumeration('TCVN_CST_RGBA_TO_YUV_422_UYVY', ETcVnColorSpaceTransform.TCVN_CST_RGBA_TO_YUV_422_UYVY);
AddLocalEnumeration('TCVN_CST_BGRA_TO_YUV_422_UYVY', ETcVnColorSpaceTransform.TCVN_CST_BGRA_TO_YUV_422_UYVY);
AddLocalEnumeration('TCVN_CST_RGBA_TO_YUV_422_Y422', ETcVnColorSpaceTransform.TCVN_CST_RGBA_TO_YUV_422_Y422);
AddLocalEnumeration('TCVN_CST_BGRA_TO_YUV_422_Y422', ETcVnColorSpaceTransform.TCVN_CST_BGRA_TO_YUV_422_Y422);
AddLocalEnumeration('TCVN_CST_RGBA_TO_YUV_422_UYNV', ETcVnColorSpaceTransform.TCVN_CST_RGBA_TO_YUV_422_UYNV);
AddLocalEnumeration('TCVN_CST_BGRA_TO_YUV_422_UYNV', ETcVnColorSpaceTransform.TCVN_CST_BGRA_TO_YUV_422_UYNV);
AddLocalEnumeration('TCVN_CST_RGB_TO_YUV_422_YUY2', ETcVnColorSpaceTransform.TCVN_CST_RGB_TO_YUV_422_YUY2);
AddLocalEnumeration('TCVN_CST_BGR_TO_YUV_422_YUY2', ETcVnColorSpaceTransform.TCVN_CST_BGR_TO_YUV_422_YUY2);
AddLocalEnumeration('TCVN_CST_RGB_TO_YUV_422_YVYU', ETcVnColorSpaceTransform.TCVN_CST_RGB_TO_YUV_422_YVYU);
AddLocalEnumeration('TCVN_CST_BGR_TO_YUV_422_YVYU', ETcVnColorSpaceTransform.TCVN_CST_BGR_TO_YUV_422_YVYU);
AddLocalEnumeration('TCVN_CST_RGB_TO_YUV_422_YUYV', ETcVnColorSpaceTransform.TCVN_CST_RGB_TO_YUV_422_YUYV);
AddLocalEnumeration('TCVN_CST_BGR_TO_YUV_422_YUYV', ETcVnColorSpaceTransform.TCVN_CST_BGR_TO_YUV_422_YUYV);
AddLocalEnumeration('TCVN_CST_RGB_TO_YUV_422_YUNV', ETcVnColorSpaceTransform.TCVN_CST_RGB_TO_YUV_422_YUNV);
AddLocalEnumeration('TCVN_CST_BGR_TO_YUV_422_YUNV', ETcVnColorSpaceTransform.TCVN_CST_BGR_TO_YUV_422_YUNV);
AddLocalEnumeration('TCVN_CST_RGBA_TO_YUV_422_YUY2', ETcVnColorSpaceTransform.TCVN_CST_RGBA_TO_YUV_422_YUY2);
AddLocalEnumeration('TCVN_CST_BGRA_TO_YUV_422_YUY2', ETcVnColorSpaceTransform.TCVN_CST_BGRA_TO_YUV_422_YUY2);
AddLocalEnumeration('TCVN_CST_RGBA_TO_YUV_422_YVYU', ETcVnColorSpaceTransform.TCVN_CST_RGBA_TO_YUV_422_YVYU);
AddLocalEnumeration('TCVN_CST_BGRA_TO_YUV_422_YVYU', ETcVnColorSpaceTransform.TCVN_CST_BGRA_TO_YUV_422_YVYU);
AddLocalEnumeration('TCVN_CST_RGBA_TO_YUV_422_YUYV', ETcVnColorSpaceTransform.TCVN_CST_RGBA_TO_YUV_422_YUYV);
AddLocalEnumeration('TCVN_CST_BGRA_TO_YUV_422_YUYV', ETcVnColorSpaceTransform.TCVN_CST_BGRA_TO_YUV_422_YUYV);
AddLocalEnumeration('TCVN_CST_RGBA_TO_YUV_422_YUNV', ETcVnColorSpaceTransform.TCVN_CST_RGBA_TO_YUV_422_YUNV);
AddLocalEnumeration('TCVN_CST_BGRA_TO_YUV_422_YUNV', ETcVnColorSpaceTransform.TCVN_CST_BGRA_TO_YUV_422_YUNV);
END_METHOD

METHOD PRIVATE AddLocalEnumeration
VAR_INPUT
	Enumeration : T_MAXSTRING;
	Value : ETcVnColorSpaceTransform;
END_VAR
AddEnumeration(Enumeration, Value);
END_METHOD

METHOD IsEnumeratorValueEqual : BOOL
VAR_INPUT
	Enumerator : I_KeyValueForwardEnumerator;
END_VAR
VAR
	storedValue : ETcVnColorSpaceTransform;
END_VAR
IF NOT Enumerator.TryGet(storedValue) THEN
	RETURN;
END_IF

IsEnumeratorValueEqual := storedValue = activeData;
END_METHOD

METHOD PUBLIC Clone : I_Datatype
VAR
    pClone : POINTER TO _ETcVnColorSpaceTransform;
END_VAR
pClone := __NEW(_ETcVnColorSpaceTransform(InitialValue := Value));
Clone := pClone^;
END_METHOD

PROPERTY PUBLIC Identifier : T_MAXSTRING
GET
Identifier := 'ETcVnColorSpaceTransform';
END_GET
END_PROPERTY

METHOD PUBLIC MakeReferenceTo
VAR_INPUT
	ReferenceTarget : REFERENCE TO ETcVnColorSpaceTransform;
END_VAR
activeData REF= ReferenceTarget;
SetBaseDatatypeReference();
END_METHOD

METHOD TryMakeReferenceTo : BOOL
VAR_INPUT
	Target : I_Datatype;
END_VAR
VAR
	pTargetData : POINTER TO ETcVnColorSpaceTransform;
END_VAR
IF NOT IsEquivalentTo(Target) THEN
	RETURN;
END_IF

pTargetData := Target.Address;
activeData REF= pTargetData^;
SetBaseDatatypeReference();
TryMakeReferenceTo := TRUE;
END_METHOD

PROPERTY PUBLIC Value : ETcVnColorSpaceTransform
GET
Value := activeData;
END_GET
SET
activeData := Value;
END_SET
END_PROPERTY

END_FUNCTION_BLOCK

// Datatypes/Enums/_ETcVnColorTrainingMethod
{attribute 'linkalways'} 
{attribute 'no_explicit_call' := 'This FB is a CLASS and must be accessed using methods or properties'}
{attribute 'enable_dynamic_creation'}
FUNCTION_BLOCK _ETcVnColorTrainingMethod EXTENDS EnumDatatypeBase
VAR
	localData : ETcVnColorTrainingMethod;
	activeData : REFERENCE TO ETcVnColorTrainingMethod;
	enumBaseDatatype : _DINT(localData);
END_VAR

METHOD PROTECTED SetBaseDatatypeReference
VAR_INPUT
END_VAR
enumBaseDatatype.MakeReferenceTo(activeData);
END_METHOD

PROPERTY PUBLIC Address : PVOID
GET
Address := ADR(activeData);
END_GET
END_PROPERTY

METHOD PUBLIC ClearReference
VAR_INPUT
END_VAR
activeData REF= localData;
SetBaseDatatypeReference();
END_METHOD

PROPERTY PUBLIC Size : UDINT
GET
Size := SIZEOF(activeData);
END_GET
END_PROPERTY

METHOD FB_init : BOOL
VAR_INPUT
	bInitRetains : BOOL; // if TRUE, the retain variables are initialized (warm start / cold start)
	bInCopyCode : BOOL;  // if TRUE, the instance afterwards gets moved into the copy code (online change)
	InitialValue : ETcVnColorTrainingMethod;
END_VAR
localData := InitialValue;
AddBaseDatatype(enumBaseDatatype);
ClearReference();

AddLocalEnumeration('TCVN_CTM_LAB', ETcVnColorTrainingMethod.TCVN_CTM_LAB);
AddLocalEnumeration('TCVN_CTM_RGB', ETcVnColorTrainingMethod.TCVN_CTM_RGB);
END_METHOD

METHOD PRIVATE AddLocalEnumeration
VAR_INPUT
	Enumeration : T_MAXSTRING;
	Value : ETcVnColorTrainingMethod;
END_VAR
AddEnumeration(Enumeration, Value);
END_METHOD

METHOD IsEnumeratorValueEqual : BOOL
VAR_INPUT
	Enumerator : I_KeyValueForwardEnumerator;
END_VAR
VAR
	storedValue : ETcVnColorTrainingMethod;
END_VAR
IF NOT Enumerator.TryGet(storedValue) THEN
	RETURN;
END_IF

IsEnumeratorValueEqual := storedValue = activeData;
END_METHOD

METHOD PUBLIC Clone : I_Datatype
VAR
    pClone : POINTER TO _ETcVnColorTrainingMethod;
END_VAR
pClone := __NEW(_ETcVnColorTrainingMethod(InitialValue := Value));
Clone := pClone^;
END_METHOD

PROPERTY PUBLIC Identifier : T_MAXSTRING
GET
Identifier := 'ETcVnColorTrainingMethod';
END_GET
END_PROPERTY

METHOD PUBLIC MakeReferenceTo
VAR_INPUT
	ReferenceTarget : REFERENCE TO ETcVnColorTrainingMethod;
END_VAR
activeData REF= ReferenceTarget;
SetBaseDatatypeReference();
END_METHOD

METHOD TryMakeReferenceTo : BOOL
VAR_INPUT
	Target : I_Datatype;
END_VAR
VAR
	pTargetData : POINTER TO ETcVnColorTrainingMethod;
END_VAR
IF NOT IsEquivalentTo(Target) THEN
	RETURN;
END_IF

pTargetData := Target.Address;
activeData REF= pTargetData^;
SetBaseDatatypeReference();
TryMakeReferenceTo := TRUE;
END_METHOD

PROPERTY PUBLIC Value : ETcVnColorTrainingMethod
GET
Value := activeData;
END_GET
SET
activeData := Value;
END_SET
END_PROPERTY

END_FUNCTION_BLOCK

// Datatypes/Enums/_ETcVnComparisonOperator
{attribute 'linkalways'}
{attribute 'no_explicit_call' := 'This FB is a CLASS and must be accessed using methods or properties'}
{attribute 'enable_dynamic_creation'}
FUNCTION_BLOCK _ETcVnComparisonOperator EXTENDS EnumDatatypeBase
VAR
	localData : ETcVnComparisonOperator;
	activeData : REFERENCE TO ETcVnComparisonOperator;
	enumBaseDatatype : _INT(localData);
END_VAR

METHOD PROTECTED SetBaseDatatypeReference
VAR_INPUT
END_VAR
enumBaseDatatype.MakeReferenceTo(activeData);
END_METHOD

PROPERTY PUBLIC Address : PVOID
GET
Address := ADR(activeData);
END_GET
END_PROPERTY

METHOD PUBLIC ClearReference
VAR_INPUT
END_VAR
activeData REF= localData;
SetBaseDatatypeReference();
END_METHOD

PROPERTY PUBLIC Size : UDINT
GET
Size := SIZEOF(activeData);
END_GET
END_PROPERTY

METHOD FB_init : BOOL
VAR_INPUT
	bInitRetains : BOOL; // if TRUE, the retain variables are initialized (warm start / cold start)
	bInCopyCode : BOOL;  // if TRUE, the instance afterwards gets moved into the copy code (online change)
	InitialValue : ETcVnComparisonOperator;
END_VAR
localData := InitialValue;
AddBaseDatatype(enumBaseDatatype);
ClearReference();

AddLocalEnumeration('TCVN_CO_LESS', ETcVnComparisonOperator.TCVN_CO_LESS);
AddLocalEnumeration('TCVN_CO_GREATER', ETcVnComparisonOperator.TCVN_CO_GREATER);
END_METHOD

METHOD PRIVATE AddLocalEnumeration
VAR_INPUT
	Enumeration : T_MAXSTRING;
	Value : ETcVnComparisonOperator;
END_VAR
AddEnumeration(Enumeration, Value);
END_METHOD

METHOD IsEnumeratorValueEqual : BOOL
VAR_INPUT
	Enumerator : I_KeyValueForwardEnumerator;
END_VAR
VAR
	storedValue : ETcVnComparisonOperator;
END_VAR
IF NOT Enumerator.TryGet(storedValue) THEN
	RETURN;
END_IF

IsEnumeratorValueEqual := storedValue = activeData;
END_METHOD

METHOD PUBLIC Clone : I_Datatype
VAR
    pClone : POINTER TO _ETcVnComparisonOperator;
END_VAR
pClone := __NEW(_ETcVnComparisonOperator(InitialValue := Value));
IF pClone = 0 THEN
    RETURN;
END_IF
Clone := pClone^;
END_METHOD

PROPERTY PUBLIC Identifier : T_MAXSTRING
GET
Identifier := 'ETcVnComparisonOperator';
END_GET
END_PROPERTY

METHOD PUBLIC MakeReferenceTo
VAR_INPUT
	ReferenceTarget : REFERENCE TO ETcVnComparisonOperator;
END_VAR
activeData REF= ReferenceTarget;
SetBaseDatatypeReference();
END_METHOD

METHOD TryMakeReferenceTo : BOOL
VAR_INPUT
	Target : I_Datatype;
END_VAR
VAR
	pTargetData : POINTER TO ETcVnComparisonOperator;
END_VAR
IF NOT IsEquivalentTo(Target) THEN
	RETURN;
END_IF

pTargetData := Target.Address;
activeData REF= pTargetData^;
SetBaseDatatypeReference();
TryMakeReferenceTo := TRUE;
END_METHOD

PROPERTY PUBLIC Value : ETcVnComparisonOperator
GET
Value := activeData;
END_GET
SET
activeData := Value;
END_SET
END_PROPERTY

END_FUNCTION_BLOCK

// Datatypes/Enums/_ETcVnConnectedComponentsAlgorithm
{attribute 'linkalways'} 
{attribute 'no_explicit_call' := 'This FB is a CLASS and must be accessed using methods or properties'}
{attribute 'enable_dynamic_creation'}
FUNCTION_BLOCK _ETcVnConnectedComponentsAlgorithm EXTENDS EnumDatatypeBase
VAR
	localData : ETcVnConnectedComponentsAlgorithm;
	activeData : REFERENCE TO ETcVnConnectedComponentsAlgorithm;
	enumBaseDatatype : _DINT(localData);
END_VAR

METHOD PROTECTED SetBaseDatatypeReference
VAR_INPUT
END_VAR
enumBaseDatatype.MakeReferenceTo(activeData);
END_METHOD

PROPERTY PUBLIC Address : PVOID
GET
Address := ADR(activeData);
END_GET
END_PROPERTY

METHOD PUBLIC ClearReference
VAR_INPUT
END_VAR
activeData REF= localData;
SetBaseDatatypeReference();
END_METHOD

PROPERTY PUBLIC Size : UDINT
GET
Size := SIZEOF(activeData);
END_GET
END_PROPERTY

METHOD FB_init : BOOL
VAR_INPUT
	bInitRetains : BOOL; // if TRUE, the retain variables are initialized (warm start / cold start)
	bInCopyCode : BOOL;  // if TRUE, the instance afterwards gets moved into the copy code (online change)
	InitialValue : ETcVnConnectedComponentsAlgorithm;
END_VAR
localData := InitialValue;
AddBaseDatatype(enumBaseDatatype);
ClearReference();

AddLocalEnumeration('TCVN_CCA_WU', ETcVnConnectedComponentsAlgorithm.TCVN_CCA_WU);
AddLocalEnumeration('TCVN_CCA_GRANA', ETcVnConnectedComponentsAlgorithm.TCVN_CCA_GRANA);
END_METHOD

METHOD PRIVATE AddLocalEnumeration
VAR_INPUT
	Enumeration : T_MAXSTRING;
	Value : ETcVnConnectedComponentsAlgorithm;
END_VAR
AddEnumeration(Enumeration, Value);
END_METHOD

METHOD IsEnumeratorValueEqual : BOOL
VAR_INPUT
	Enumerator : I_KeyValueForwardEnumerator;
END_VAR
VAR
	storedValue : ETcVnConnectedComponentsAlgorithm;
END_VAR
IF NOT Enumerator.TryGet(storedValue) THEN
	RETURN;
END_IF

IsEnumeratorValueEqual := storedValue = activeData;
END_METHOD

METHOD PUBLIC Clone : I_Datatype
VAR
    pClone : POINTER TO _ETcVnConnectedComponentsAlgorithm;
END_VAR
pClone := __NEW(_ETcVnConnectedComponentsAlgorithm(InitialValue := Value));
Clone := pClone^;
END_METHOD

PROPERTY PUBLIC Identifier : T_MAXSTRING
GET
Identifier := 'ETcVnConnectedComponentsAlgorithm';
END_GET
END_PROPERTY

METHOD PUBLIC MakeReferenceTo
VAR_INPUT
	ReferenceTarget : REFERENCE TO ETcVnConnectedComponentsAlgorithm;
END_VAR
activeData REF= ReferenceTarget;
SetBaseDatatypeReference();
END_METHOD

METHOD TryMakeReferenceTo : BOOL
VAR_INPUT
	Target : I_Datatype;
END_VAR
VAR
	pTargetData : POINTER TO ETcVnConnectedComponentsAlgorithm;
END_VAR
IF NOT IsEquivalentTo(Target) THEN
	RETURN;
END_IF

pTargetData := Target.Address;
activeData REF= pTargetData^;
SetBaseDatatypeReference();
TryMakeReferenceTo := TRUE;
END_METHOD

PROPERTY PUBLIC Value : ETcVnConnectedComponentsAlgorithm
GET
Value := activeData;
END_GET
SET
activeData := Value;
END_SET
END_PROPERTY

END_FUNCTION_BLOCK

// Datatypes/Enums/_ETcVnContainerExportFormat
{attribute 'linkalways'} 
{attribute 'no_explicit_call' := 'This FB is a CLASS and must be accessed using methods or properties'}
{attribute 'enable_dynamic_creation'}
FUNCTION_BLOCK _ETcVnContainerExportFormat EXTENDS EnumDatatypeBase
VAR
	localData : ETcVnContainerExportFormat;
	activeData : REFERENCE TO ETcVnContainerExportFormat;
	enumBaseDatatype : _UINT(localData);
END_VAR

METHOD PROTECTED SetBaseDatatypeReference
VAR_INPUT
END_VAR
enumBaseDatatype.MakeReferenceTo(activeData);
END_METHOD

PROPERTY PUBLIC Address : PVOID
GET
Address := ADR(activeData);
END_GET
END_PROPERTY

METHOD PUBLIC ClearReference
VAR_INPUT
END_VAR
activeData REF= localData;
SetBaseDatatypeReference();
END_METHOD

PROPERTY PUBLIC Size : UDINT
GET
Size := SIZEOF(activeData);
END_GET
END_PROPERTY

METHOD FB_init : BOOL
VAR_INPUT
	bInitRetains : BOOL; // if TRUE, the retain variables are initialized (warm start / cold start)
	bInCopyCode : BOOL;  // if TRUE, the instance afterwards gets moved into the copy code (online change)
	InitialValue : ETcVnContainerExportFormat;
END_VAR
localData := InitialValue;
AddBaseDatatype(enumBaseDatatype);
ClearReference();

AddLocalEnumeration('TCVN_CEF_XML', ETcVnContainerExportFormat.TCVN_CEF_XML);
AddLocalEnumeration('TCVN_CEF_XML_SERIALIZED', ETcVnContainerExportFormat.TCVN_CEF_XML_SERIALIZED);
AddLocalEnumeration('TCVN_CEF_CSV', ETcVnContainerExportFormat.TCVN_CEF_CSV);
AddLocalEnumeration('TCVN_CEF_BINARY', ETcVnContainerExportFormat.TCVN_CEF_BINARY);
END_METHOD

METHOD PRIVATE AddLocalEnumeration
VAR_INPUT
	Enumeration : T_MAXSTRING;
	Value : ETcVnContainerExportFormat;
END_VAR
AddEnumeration(Enumeration, Value);
END_METHOD

METHOD IsEnumeratorValueEqual : BOOL
VAR_INPUT
	Enumerator : I_KeyValueForwardEnumerator;
END_VAR
VAR
	storedValue : ETcVnContainerExportFormat;
END_VAR
IF NOT Enumerator.TryGet(storedValue) THEN
	RETURN;
END_IF

IsEnumeratorValueEqual := storedValue = activeData;
END_METHOD

METHOD PUBLIC Clone : I_Datatype
VAR
    pClone : POINTER TO _ETcVnContainerExportFormat;
END_VAR
pClone := __NEW(_ETcVnContainerExportFormat(InitialValue := Value));
Clone := pClone^;
END_METHOD

PROPERTY PUBLIC Identifier : T_MAXSTRING
GET
Identifier := 'ETcVnContainerExportFormat';
END_GET
END_PROPERTY

METHOD PUBLIC MakeReferenceTo
VAR_INPUT
	ReferenceTarget : REFERENCE TO ETcVnContainerExportFormat;
END_VAR
activeData REF= ReferenceTarget;
SetBaseDatatypeReference();
END_METHOD

METHOD TryMakeReferenceTo : BOOL
VAR_INPUT
	Target : I_Datatype;
END_VAR
VAR
	pTargetData : POINTER TO ETcVnContainerExportFormat;
END_VAR
IF NOT IsEquivalentTo(Target) THEN
	RETURN;
END_IF

pTargetData := Target.Address;
activeData REF= pTargetData^;
SetBaseDatatypeReference();
TryMakeReferenceTo := TRUE;
END_METHOD

PROPERTY PUBLIC Value : ETcVnContainerExportFormat
GET
Value := activeData;
END_GET
SET
activeData := Value;
END_SET
END_PROPERTY

END_FUNCTION_BLOCK

// Datatypes/Enums/_ETcVnContourApproximationMethod
{attribute 'linkalways'} 
{attribute 'no_explicit_call' := 'This FB is a CLASS and must be accessed using methods or properties'}
{attribute 'enable_dynamic_creation'}
FUNCTION_BLOCK _ETcVnContourApproximationMethod EXTENDS EnumDatatypeBase
VAR
	localData : ETcVnContourApproximationMethod;
	activeData : REFERENCE TO ETcVnContourApproximationMethod;
	enumBaseDatatype : _DINT(localData);
END_VAR

METHOD PROTECTED SetBaseDatatypeReference
VAR_INPUT
END_VAR
enumBaseDatatype.MakeReferenceTo(activeData);
END_METHOD

PROPERTY PUBLIC Address : PVOID
GET
Address := ADR(activeData);
END_GET
END_PROPERTY

METHOD PUBLIC ClearReference
VAR_INPUT
END_VAR
activeData REF= localData;
SetBaseDatatypeReference();
END_METHOD

PROPERTY PUBLIC Size : UDINT
GET
Size := SIZEOF(activeData);
END_GET
END_PROPERTY

METHOD FB_init : BOOL
VAR_INPUT
	bInitRetains : BOOL; // if TRUE, the retain variables are initialized (warm start / cold start)
	bInCopyCode : BOOL;  // if TRUE, the instance afterwards gets moved into the copy code (online change)
	InitialValue : ETcVnContourApproximationMethod;
END_VAR
localData := InitialValue;
AddBaseDatatype(enumBaseDatatype);
ClearReference();

AddLocalEnumeration('TCVN_CAM_NONE', ETcVnContourApproximationMethod.TCVN_CAM_NONE);
AddLocalEnumeration('TCVN_CAM_SIMPLE', ETcVnContourApproximationMethod.TCVN_CAM_SIMPLE);
AddLocalEnumeration('TCVN_CAM_TC89_L1', ETcVnContourApproximationMethod.TCVN_CAM_TC89_L1);
AddLocalEnumeration('TCVN_CAM_TC89_KCOS', ETcVnContourApproximationMethod.TCVN_CAM_TC89_KCOS);
END_METHOD

METHOD PRIVATE AddLocalEnumeration
VAR_INPUT
	Enumeration : T_MAXSTRING;
	Value : ETcVnContourApproximationMethod;
END_VAR
AddEnumeration(Enumeration, Value);
END_METHOD

METHOD IsEnumeratorValueEqual : BOOL
VAR_INPUT
	Enumerator : I_KeyValueForwardEnumerator;
END_VAR
VAR
	storedValue : ETcVnContourApproximationMethod;
END_VAR
IF NOT Enumerator.TryGet(storedValue) THEN
	RETURN;
END_IF

IsEnumeratorValueEqual := storedValue = activeData;
END_METHOD

METHOD PUBLIC Clone : I_Datatype
VAR
    pClone : POINTER TO _ETcVnContourApproximationMethod;
END_VAR
pClone := __NEW(_ETcVnContourApproximationMethod(InitialValue := Value));
Clone := pClone^;
END_METHOD

PROPERTY PUBLIC Identifier : T_MAXSTRING
GET
Identifier := 'ETcVnContourApproximationMethod';
END_GET
END_PROPERTY

METHOD PUBLIC MakeReferenceTo
VAR_INPUT
	ReferenceTarget : REFERENCE TO ETcVnContourApproximationMethod;
END_VAR
activeData REF= ReferenceTarget;
SetBaseDatatypeReference();
END_METHOD

METHOD TryMakeReferenceTo : BOOL
VAR_INPUT
	Target : I_Datatype;
END_VAR
VAR
	pTargetData : POINTER TO ETcVnContourApproximationMethod;
END_VAR
IF NOT IsEquivalentTo(Target) THEN
	RETURN;
END_IF

pTargetData := Target.Address;
activeData REF= pTargetData^;
SetBaseDatatypeReference();
TryMakeReferenceTo := TRUE;
END_METHOD

PROPERTY PUBLIC Value : ETcVnContourApproximationMethod
GET
Value := activeData;
END_GET
SET
activeData := Value;
END_SET
END_PROPERTY

END_FUNCTION_BLOCK

// Datatypes/Enums/_ETcVnContourRetrievalMode
{attribute 'linkalways'} 
{attribute 'no_explicit_call' := 'This FB is a CLASS and must be accessed using methods or properties'}
{attribute 'enable_dynamic_creation'}
FUNCTION_BLOCK _ETcVnContourRetrievalMode EXTENDS EnumDatatypeBase
VAR
	localData : ETcVnContourRetrievalMode;
	activeData : REFERENCE TO ETcVnContourRetrievalMode;
	enumBaseDatatype : _DINT(localData);
END_VAR

METHOD PROTECTED SetBaseDatatypeReference
VAR_INPUT
END_VAR
enumBaseDatatype.MakeReferenceTo(activeData);
END_METHOD

PROPERTY PUBLIC Address : PVOID
GET
Address := ADR(activeData);
END_GET
END_PROPERTY

METHOD PUBLIC ClearReference
VAR_INPUT
END_VAR
activeData REF= localData;
SetBaseDatatypeReference();
END_METHOD

PROPERTY PUBLIC Size : UDINT
GET
Size := SIZEOF(activeData);
END_GET
END_PROPERTY

METHOD FB_init : BOOL
VAR_INPUT
	bInitRetains : BOOL; // if TRUE, the retain variables are initialized (warm start / cold start)
	bInCopyCode : BOOL;  // if TRUE, the instance afterwards gets moved into the copy code (online change)
	InitialValue : ETcVnContourRetrievalMode;
END_VAR
localData := InitialValue;
AddBaseDatatype(enumBaseDatatype);
ClearReference();

AddLocalEnumeration('TCVN_CRM_EXTERNAL', ETcVnContourRetrievalMode.TCVN_CRM_EXTERNAL);
AddLocalEnumeration('TCVN_CRM_LIST', ETcVnContourRetrievalMode.TCVN_CRM_LIST);
AddLocalEnumeration('TCVN_CRM_CONNECTED_COMPONENTS', ETcVnContourRetrievalMode.TCVN_CRM_CONNECTED_COMPONENTS);
AddLocalEnumeration('TCVN_CRM_TREE', ETcVnContourRetrievalMode.TCVN_CRM_TREE);
AddLocalEnumeration('TCVN_CRM_FLOODFILL', ETcVnContourRetrievalMode.TCVN_CRM_FLOODFILL);
END_METHOD

METHOD PRIVATE AddLocalEnumeration
VAR_INPUT
	Enumeration : T_MAXSTRING;
	Value : ETcVnContourRetrievalMode;
END_VAR
AddEnumeration(Enumeration, Value);
END_METHOD

METHOD IsEnumeratorValueEqual : BOOL
VAR_INPUT
	Enumerator : I_KeyValueForwardEnumerator;
END_VAR
VAR
	storedValue : ETcVnContourRetrievalMode;
END_VAR
IF NOT Enumerator.TryGet(storedValue) THEN
	RETURN;
END_IF

IsEnumeratorValueEqual := storedValue = activeData;
END_METHOD

METHOD PUBLIC Clone : I_Datatype
VAR
    pClone : POINTER TO _ETcVnContourRetrievalMode;
END_VAR
pClone := __NEW(_ETcVnContourRetrievalMode(InitialValue := Value));
Clone := pClone^;
END_METHOD

PROPERTY PUBLIC Identifier : T_MAXSTRING
GET
Identifier := 'ETcVnContourRetrievalMode';
END_GET
END_PROPERTY

METHOD PUBLIC MakeReferenceTo
VAR_INPUT
	ReferenceTarget : REFERENCE TO ETcVnContourRetrievalMode;
END_VAR
activeData REF= ReferenceTarget;
SetBaseDatatypeReference();
END_METHOD

METHOD TryMakeReferenceTo : BOOL
VAR_INPUT
	Target : I_Datatype;
END_VAR
VAR
	pTargetData : POINTER TO ETcVnContourRetrievalMode;
END_VAR
IF NOT IsEquivalentTo(Target) THEN
	RETURN;
END_IF

pTargetData := Target.Address;
activeData REF= pTargetData^;
SetBaseDatatypeReference();
TryMakeReferenceTo := TRUE;
END_METHOD

PROPERTY PUBLIC Value : ETcVnContourRetrievalMode
GET
Value := activeData;
END_GET
SET
activeData := Value;
END_SET
END_PROPERTY

END_FUNCTION_BLOCK

// Datatypes/Enums/_ETcVnContoursMatchComparisonMethod
{attribute 'linkalways'} 
{attribute 'no_explicit_call' := 'This FB is a CLASS and must be accessed using methods or properties'}
{attribute 'enable_dynamic_creation'}
FUNCTION_BLOCK _ETcVnContoursMatchComparisonMethod EXTENDS EnumDatatypeBase
VAR
	localData : ETcVnContoursMatchComparisonMethod;
	activeData : REFERENCE TO ETcVnContoursMatchComparisonMethod;
	enumBaseDatatype : _DINT(localData);
END_VAR

METHOD PROTECTED SetBaseDatatypeReference
VAR_INPUT
END_VAR
enumBaseDatatype.MakeReferenceTo(activeData);
END_METHOD

PROPERTY PUBLIC Address : PVOID
GET
Address := ADR(activeData);
END_GET
END_PROPERTY

METHOD PUBLIC ClearReference
VAR_INPUT
END_VAR
activeData REF= localData;
SetBaseDatatypeReference();
END_METHOD

PROPERTY PUBLIC Size : UDINT
GET
Size := SIZEOF(activeData);
END_GET
END_PROPERTY

METHOD FB_init : BOOL
VAR_INPUT
	bInitRetains : BOOL; // if TRUE, the retain variables are initialized (warm start / cold start)
	bInCopyCode : BOOL;  // if TRUE, the instance afterwards gets moved into the copy code (online change)
	InitialValue : ETcVnContoursMatchComparisonMethod;
END_VAR
localData := InitialValue;
AddBaseDatatype(enumBaseDatatype);
ClearReference();

AddLocalEnumeration('TCVN_CMCM_CONTOURS_MATCH_I1', ETcVnContoursMatchComparisonMethod.TCVN_CMCM_CONTOURS_MATCH_I1);
AddLocalEnumeration('TCVN_CMCM_CONTOURS_MATCH_I2', ETcVnContoursMatchComparisonMethod.TCVN_CMCM_CONTOURS_MATCH_I2);
AddLocalEnumeration('TCVN_CMCM_CONTOURS_MATCH_I3', ETcVnContoursMatchComparisonMethod.TCVN_CMCM_CONTOURS_MATCH_I3);
END_METHOD

METHOD PRIVATE AddLocalEnumeration
VAR_INPUT
	Enumeration : T_MAXSTRING;
	Value : ETcVnContoursMatchComparisonMethod;
END_VAR
AddEnumeration(Enumeration, Value);
END_METHOD

METHOD IsEnumeratorValueEqual : BOOL
VAR_INPUT
	Enumerator : I_KeyValueForwardEnumerator;
END_VAR
VAR
	storedValue : ETcVnContoursMatchComparisonMethod;
END_VAR
IF NOT Enumerator.TryGet(storedValue) THEN
	RETURN;
END_IF

IsEnumeratorValueEqual := storedValue = activeData;
END_METHOD

METHOD PUBLIC Clone : I_Datatype
VAR
    pClone : POINTER TO _ETcVnContoursMatchComparisonMethod;
END_VAR
pClone := __NEW(_ETcVnContoursMatchComparisonMethod(InitialValue := Value));
Clone := pClone^;
END_METHOD

PROPERTY PUBLIC Identifier : T_MAXSTRING
GET
Identifier := 'ETcVnContoursMatchComparisonMethod';
END_GET
END_PROPERTY

METHOD PUBLIC MakeReferenceTo
VAR_INPUT
	ReferenceTarget : REFERENCE TO ETcVnContoursMatchComparisonMethod;
END_VAR
activeData REF= ReferenceTarget;
SetBaseDatatypeReference();
END_METHOD

METHOD TryMakeReferenceTo : BOOL
VAR_INPUT
	Target : I_Datatype;
END_VAR
VAR
	pTargetData : POINTER TO ETcVnContoursMatchComparisonMethod;
END_VAR
IF NOT IsEquivalentTo(Target) THEN
	RETURN;
END_IF

pTargetData := Target.Address;
activeData REF= pTargetData^;
SetBaseDatatypeReference();
TryMakeReferenceTo := TRUE;
END_METHOD

PROPERTY PUBLIC Value : ETcVnContoursMatchComparisonMethod
GET
Value := activeData;
END_GET
SET
activeData := Value;
END_SET
END_PROPERTY

END_FUNCTION_BLOCK

// Datatypes/Enums/_ETcVnDataLayout
{attribute 'linkalways'} 
{attribute 'no_explicit_call' := 'This FB is a CLASS and must be accessed using methods or properties'}
{attribute 'enable_dynamic_creation'}
FUNCTION_BLOCK _ETcVnDataLayout EXTENDS EnumDatatypeBase
VAR
	localData : ETcVnDataLayout;
	activeData : REFERENCE TO ETcVnDataLayout;
	enumBaseDatatype : _ULINT(localData);
END_VAR

METHOD PROTECTED SetBaseDatatypeReference
VAR_INPUT
END_VAR
enumBaseDatatype.MakeReferenceTo(activeData);
END_METHOD

PROPERTY PUBLIC Address : PVOID
GET
Address := ADR(activeData);
END_GET
END_PROPERTY

METHOD PUBLIC ClearReference
VAR_INPUT
END_VAR
activeData REF= localData;
SetBaseDatatypeReference();
END_METHOD

PROPERTY PUBLIC Size : UDINT
GET
Size := SIZEOF(activeData);
END_GET
END_PROPERTY

METHOD FB_init : BOOL
VAR_INPUT
	bInitRetains : BOOL; // if TRUE, the retain variables are initialized (warm start / cold start)
	bInCopyCode : BOOL;  // if TRUE, the instance afterwards gets moved into the copy code (online change)
	InitialValue : ETcVnDataLayout;
END_VAR
localData := InitialValue;
AddBaseDatatype(enumBaseDatatype);
ClearReference();

AddLocalEnumeration('TCVN_DL_DEFAULT', ETcVnDataLayout.TCVN_DL_DEFAULT);
AddLocalEnumeration('TCVN_DL_2D_HW', ETcVnDataLayout.TCVN_DL_2D_HW);
AddLocalEnumeration('TCVN_DL_2D_WH', ETcVnDataLayout.TCVN_DL_2D_WH);
AddLocalEnumeration('TCVN_DL_3D_CHW', ETcVnDataLayout.TCVN_DL_3D_CHW);
AddLocalEnumeration('TCVN_DL_3D_HWC', ETcVnDataLayout.TCVN_DL_3D_HWC);
AddLocalEnumeration('TCVN_DL_4D_NCHW', ETcVnDataLayout.TCVN_DL_4D_NCHW);
AddLocalEnumeration('TCVN_DL_4D_NHWC', ETcVnDataLayout.TCVN_DL_4D_NHWC);
END_METHOD

METHOD PRIVATE AddLocalEnumeration
VAR_INPUT
	Enumeration : T_MAXSTRING;
	Value : ETcVnDataLayout;
END_VAR
AddEnumeration(Enumeration, Value);
END_METHOD

METHOD IsEnumeratorValueEqual : BOOL
VAR_INPUT
	Enumerator : I_KeyValueForwardEnumerator;
END_VAR
VAR
	storedValue : ETcVnDataLayout;
END_VAR
IF NOT Enumerator.TryGet(storedValue) THEN
	RETURN;
END_IF

IsEnumeratorValueEqual := storedValue = activeData;
END_METHOD

METHOD PUBLIC Clone : I_Datatype
VAR
    pClone : POINTER TO _ETcVnDataLayout;
END_VAR
pClone := __NEW(_ETcVnDataLayout(InitialValue := Value));
Clone := pClone^;
END_METHOD

PROPERTY PUBLIC Identifier : T_MAXSTRING
GET
Identifier := 'ETcVnDataLayout';
END_GET
END_PROPERTY

METHOD PUBLIC MakeReferenceTo
VAR_INPUT
	ReferenceTarget : REFERENCE TO ETcVnDataLayout;
END_VAR
activeData REF= ReferenceTarget;
SetBaseDatatypeReference();
END_METHOD

METHOD TryMakeReferenceTo : BOOL
VAR_INPUT
	Target : I_Datatype;
END_VAR
VAR
	pTargetData : POINTER TO ETcVnDataLayout;
END_VAR
IF NOT IsEquivalentTo(Target) THEN
	RETURN;
END_IF

pTargetData := Target.Address;
activeData REF= pTargetData^;
SetBaseDatatypeReference();
TryMakeReferenceTo := TRUE;
END_METHOD

PROPERTY PUBLIC Value : ETcVnDataLayout
GET
Value := activeData;
END_GET
SET
activeData := Value;
END_SET
END_PROPERTY

END_FUNCTION_BLOCK

// Datatypes/Enums/_ETcVnDataMatrixOptions
{attribute 'linkalways'} 
{attribute 'no_explicit_call' := 'This FB is a CLASS and must be accessed using methods or properties'}
{attribute 'enable_dynamic_creation'}
FUNCTION_BLOCK _ETcVnDataMatrixOptions EXTENDS EnumDatatypeBase
VAR
	localData : ETcVnDataMatrixOptions;
	activeData : REFERENCE TO ETcVnDataMatrixOptions;
	enumBaseDatatype : _ULINT(localData);
END_VAR

METHOD PROTECTED SetBaseDatatypeReference
VAR_INPUT
END_VAR
enumBaseDatatype.MakeReferenceTo(activeData);
END_METHOD

PROPERTY PUBLIC Address : PVOID
GET
Address := ADR(activeData);
END_GET
END_PROPERTY

METHOD PUBLIC ClearReference
VAR_INPUT
END_VAR
activeData REF= localData;
SetBaseDatatypeReference();
END_METHOD

PROPERTY PUBLIC Size : UDINT
GET
Size := SIZEOF(activeData);
END_GET
END_PROPERTY

METHOD FB_init : BOOL
VAR_INPUT
	bInitRetains : BOOL; // if TRUE, the retain variables are initialized (warm start / cold start)
	bInCopyCode : BOOL;  // if TRUE, the instance afterwards gets moved into the copy code (online change)
	InitialValue : ETcVnDataMatrixOptions;
END_VAR
localData := InitialValue;
AddBaseDatatype(enumBaseDatatype);
ClearReference();

AddLocalEnumeration('TCVN_DMO_DEFAULT', ETcVnDataMatrixOptions.TCVN_DMO_DEFAULT);
AddLocalEnumeration('TCVN_DMO_BINARY_INPUT', ETcVnDataMatrixOptions.TCVN_DMO_BINARY_INPUT);
AddLocalEnumeration('TCVN_DMO_GLOBAL_THRESHOLD', ETcVnDataMatrixOptions.TCVN_DMO_GLOBAL_THRESHOLD);
AddLocalEnumeration('TCVN_DMO_BINARY_GRID', ETcVnDataMatrixOptions.TCVN_DMO_BINARY_GRID);
AddLocalEnumeration('TCVN_DMO_STATIC_GRID', ETcVnDataMatrixOptions.TCVN_DMO_STATIC_GRID);
AddLocalEnumeration('TCVN_DMO_REGULAR_COLOR', ETcVnDataMatrixOptions.TCVN_DMO_REGULAR_COLOR);
AddLocalEnumeration('TCVN_DMO_INVERTED_COLOR', ETcVnDataMatrixOptions.TCVN_DMO_INVERTED_COLOR);
END_METHOD

METHOD PRIVATE AddLocalEnumeration
VAR_INPUT
	Enumeration : T_MAXSTRING;
	Value : ETcVnDataMatrixOptions;
END_VAR
AddEnumeration(Enumeration, Value);
END_METHOD

METHOD IsEnumeratorValueEqual : BOOL
VAR_INPUT
	Enumerator : I_KeyValueForwardEnumerator;
END_VAR
VAR
	storedValue : ETcVnDataMatrixOptions;
END_VAR
IF NOT Enumerator.TryGet(storedValue) THEN
	RETURN;
END_IF

IsEnumeratorValueEqual := storedValue = activeData;
END_METHOD

METHOD PUBLIC Clone : I_Datatype
VAR
    pClone : POINTER TO _ETcVnDataMatrixOptions;
END_VAR
pClone := __NEW(_ETcVnDataMatrixOptions(InitialValue := Value));
Clone := pClone^;
END_METHOD

PROPERTY PUBLIC Identifier : T_MAXSTRING
GET
Identifier := 'ETcVnDataMatrixOptions';
END_GET
END_PROPERTY

METHOD PUBLIC MakeReferenceTo
VAR_INPUT
	ReferenceTarget : REFERENCE TO ETcVnDataMatrixOptions;
END_VAR
activeData REF= ReferenceTarget;
SetBaseDatatypeReference();
END_METHOD

METHOD TryMakeReferenceTo : BOOL
VAR_INPUT
	Target : I_Datatype;
END_VAR
VAR
	pTargetData : POINTER TO ETcVnDataMatrixOptions;
END_VAR
IF NOT IsEquivalentTo(Target) THEN
	RETURN;
END_IF

pTargetData := Target.Address;
activeData REF= pTargetData^;
SetBaseDatatypeReference();
TryMakeReferenceTo := TRUE;
END_METHOD

PROPERTY PUBLIC Value : ETcVnDataMatrixOptions
GET
Value := activeData;
END_GET
SET
activeData := Value;
END_SET
END_PROPERTY

END_FUNCTION_BLOCK

// Datatypes/Enums/_ETcVnDetectBarcodesWalshOptions
{attribute 'linkalways'}
{attribute 'no_explicit_call' := 'This FB is a CLASS and must be accessed using methods or properties'}
{attribute 'enable_dynamic_creation'}
FUNCTION_BLOCK _ETcVnDetectBarcodesWalshOptions EXTENDS EnumDatatypeBase
VAR
	localData : ETcVnDetectBarcodesWalshOptions;
	activeData : REFERENCE TO ETcVnDetectBarcodesWalshOptions;
	enumBaseDatatype : _UDINT(localData);
END_VAR

METHOD PROTECTED SetBaseDatatypeReference
VAR_INPUT
END_VAR
enumBaseDatatype.MakeReferenceTo(activeData);
END_METHOD

PROPERTY PUBLIC Address : PVOID
GET
Address := ADR(activeData);
END_GET
END_PROPERTY

METHOD PUBLIC ClearReference
VAR_INPUT
END_VAR
activeData REF= localData;
SetBaseDatatypeReference();
END_METHOD

PROPERTY PUBLIC Size : UDINT
GET
Size := SIZEOF(activeData);
END_GET
END_PROPERTY

METHOD FB_init : BOOL
VAR_INPUT
	bInitRetains : BOOL; // if TRUE, the retain variables are initialized (warm start / cold start)
	bInCopyCode : BOOL;  // if TRUE, the instance afterwards gets moved into the copy code (online change)
	InitialValue : ETcVnDetectBarcodesWalshOptions;
END_VAR
localData := InitialValue;
AddBaseDatatype(enumBaseDatatype);
ClearReference();

AddLocalEnumeration('TCVN_DBWO_HORIZONTAL', ETcVnDetectBarcodesWalshOptions.TCVN_DBWO_HORIZONTAL);
AddLocalEnumeration('TCVN_DBWO_VERTICAL', ETcVnDetectBarcodesWalshOptions.TCVN_DBWO_VERTICAL);
AddLocalEnumeration('TCVN_DBWO_DIAGONAL_45', ETcVnDetectBarcodesWalshOptions.TCVN_DBWO_DIAGONAL_45);
AddLocalEnumeration('TCVN_DBWO_DIAGONAL_135', ETcVnDetectBarcodesWalshOptions.TCVN_DBWO_DIAGONAL_135);
AddLocalEnumeration('TCVN_DBWO_ALL_DIRECTIONS', ETcVnDetectBarcodesWalshOptions.TCVN_DBWO_ALL_DIRECTIONS);
END_METHOD

METHOD PRIVATE AddLocalEnumeration
VAR_INPUT
	Enumeration : T_MAXSTRING;
	Value : ETcVnDetectBarcodesWalshOptions;
END_VAR
AddEnumeration(Enumeration, Value);
END_METHOD

METHOD IsEnumeratorValueEqual : BOOL
VAR_INPUT
	Enumerator : I_KeyValueForwardEnumerator;
END_VAR
VAR
	storedValue : ETcVnDetectBarcodesWalshOptions;
END_VAR
IF NOT Enumerator.TryGet(storedValue) THEN
	RETURN;
END_IF

IsEnumeratorValueEqual := storedValue = activeData;
END_METHOD

METHOD PUBLIC Clone : I_Datatype
VAR
    pClone : POINTER TO _ETcVnDetectBarcodesWalshOptions;
END_VAR
pClone := __NEW(_ETcVnDetectBarcodesWalshOptions(InitialValue := Value));
IF pClone = 0 THEN
    RETURN;
END_IF
Clone := pClone^;
END_METHOD

PROPERTY PUBLIC Identifier : T_MAXSTRING
GET
Identifier := 'ETcVnDetectBarcodesWalshOptions';
END_GET
END_PROPERTY

METHOD PUBLIC MakeReferenceTo
VAR_INPUT
	ReferenceTarget : REFERENCE TO ETcVnDetectBarcodesWalshOptions;
END_VAR
activeData REF= ReferenceTarget;
SetBaseDatatypeReference();
END_METHOD

METHOD TryMakeReferenceTo : BOOL
VAR_INPUT
	Target : I_Datatype;
END_VAR
VAR
	pTargetData : POINTER TO ETcVnDetectBarcodesWalshOptions;
END_VAR
IF NOT IsEquivalentTo(Target) THEN
	RETURN;
END_IF

pTargetData := Target.Address;
activeData REF= pTargetData^;
SetBaseDatatypeReference();
TryMakeReferenceTo := TRUE;
END_METHOD

PROPERTY PUBLIC Value : ETcVnDetectBarcodesWalshOptions
GET
Value := activeData;
END_GET
SET
activeData := Value;
END_SET
END_PROPERTY

END_FUNCTION_BLOCK

// Datatypes/Enums/_ETcVnDetectPatternPointsOptions
{attribute 'linkalways'}
{attribute 'no_explicit_call' := 'This FB is a CLASS and must be accessed using methods or properties'}
{attribute 'enable_dynamic_creation'}
FUNCTION_BLOCK _ETcVnDetectPatternPointsOptions EXTENDS EnumDatatypeBase
VAR
	localData : ETcVnDetectPatternPointsOptions;
	activeData : REFERENCE TO ETcVnDetectPatternPointsOptions;
	enumBaseDatatype : _UDINT(localData);
END_VAR

METHOD PROTECTED SetBaseDatatypeReference
VAR_INPUT
END_VAR
enumBaseDatatype.MakeReferenceTo(activeData);
END_METHOD

PROPERTY PUBLIC Address : PVOID
GET
Address := ADR(activeData);
END_GET
END_PROPERTY

METHOD PUBLIC ClearReference
VAR_INPUT
END_VAR
activeData REF= localData;
SetBaseDatatypeReference();
END_METHOD

PROPERTY PUBLIC Size : UDINT
GET
Size := SIZEOF(activeData);
END_GET
END_PROPERTY

METHOD FB_init : BOOL
VAR_INPUT
	bInitRetains : BOOL; // if TRUE, the retain variables are initialized (warm start / cold start)
	bInCopyCode : BOOL;  // if TRUE, the instance afterwards gets moved into the copy code (online change)
	InitialValue : ETcVnDetectPatternPointsOptions;
END_VAR
localData := InitialValue;
AddBaseDatatype(enumBaseDatatype);
ClearReference();

AddLocalEnumeration('TCVN_DPPO_SYMMETRIC', ETcVnDetectPatternPointsOptions.TCVN_DPPO_SYMMETRIC);
AddLocalEnumeration('TCVN_DPPO_ASYMMETRIC', ETcVnDetectPatternPointsOptions.TCVN_DPPO_ASYMMETRIC);
AddLocalEnumeration('TCVN_DPPO_CLUSTERING', ETcVnDetectPatternPointsOptions.TCVN_DPPO_CLUSTERING);
END_METHOD

METHOD PRIVATE AddLocalEnumeration
VAR_INPUT
	Enumeration : T_MAXSTRING;
	Value : ETcVnDetectPatternPointsOptions;
END_VAR
AddEnumeration(Enumeration, Value);
END_METHOD

METHOD IsEnumeratorValueEqual : BOOL
VAR_INPUT
	Enumerator : I_KeyValueForwardEnumerator;
END_VAR
VAR
	storedValue : ETcVnDetectPatternPointsOptions;
END_VAR
IF NOT Enumerator.TryGet(storedValue) THEN
	RETURN;
END_IF

IsEnumeratorValueEqual := storedValue = activeData;
END_METHOD

METHOD PUBLIC Clone : I_Datatype
VAR
    pClone : POINTER TO _ETcVnDetectPatternPointsOptions;
END_VAR
pClone := __NEW(_ETcVnDetectPatternPointsOptions(InitialValue := Value));
IF pClone = 0 THEN
    RETURN;
END_IF
Clone := pClone^;
END_METHOD

PROPERTY PUBLIC Identifier : T_MAXSTRING
GET
Identifier := 'ETcVnDetectPatternPointsOptions';
END_GET
END_PROPERTY

METHOD PUBLIC MakeReferenceTo
VAR_INPUT
	ReferenceTarget : REFERENCE TO ETcVnDetectPatternPointsOptions;
END_VAR
activeData REF= ReferenceTarget;
SetBaseDatatypeReference();
END_METHOD

METHOD TryMakeReferenceTo : BOOL
VAR_INPUT
	Target : I_Datatype;
END_VAR
VAR
	pTargetData : POINTER TO ETcVnDetectPatternPointsOptions;
END_VAR
IF NOT IsEquivalentTo(Target) THEN
	RETURN;
END_IF

pTargetData := Target.Address;
activeData REF= pTargetData^;
SetBaseDatatypeReference();
TryMakeReferenceTo := TRUE;
END_METHOD

PROPERTY PUBLIC Value : ETcVnDetectPatternPointsOptions
GET
Value := activeData;
END_GET
SET
activeData := Value;
END_SET
END_PROPERTY

END_FUNCTION_BLOCK

// Datatypes/Enums/_ETcVnDiffusivityTypeKAZE
{attribute 'linkalways'} 
{attribute 'no_explicit_call' := 'This FB is a CLASS and must be accessed using methods or properties'}
{attribute 'enable_dynamic_creation'}
FUNCTION_BLOCK _ETcVnDiffusivityTypeKAZE EXTENDS EnumDatatypeBase
VAR
	localData : ETcVnDiffusivityTypeKAZE;
	activeData : REFERENCE TO ETcVnDiffusivityTypeKAZE;
	enumBaseDatatype : _DINT(localData);
END_VAR

METHOD PROTECTED SetBaseDatatypeReference
VAR_INPUT
END_VAR
enumBaseDatatype.MakeReferenceTo(activeData);
END_METHOD

PROPERTY PUBLIC Address : PVOID
GET
Address := ADR(activeData);
END_GET
END_PROPERTY

METHOD PUBLIC ClearReference
VAR_INPUT
END_VAR
activeData REF= localData;
SetBaseDatatypeReference();
END_METHOD

PROPERTY PUBLIC Size : UDINT
GET
Size := SIZEOF(activeData);
END_GET
END_PROPERTY

METHOD FB_init : BOOL
VAR_INPUT
	bInitRetains : BOOL; // if TRUE, the retain variables are initialized (warm start / cold start)
	bInCopyCode : BOOL;  // if TRUE, the instance afterwards gets moved into the copy code (online change)
	InitialValue : ETcVnDiffusivityTypeKAZE;
END_VAR
localData := InitialValue;
AddBaseDatatype(enumBaseDatatype);
ClearReference();

AddLocalEnumeration('TCVN_DT1_KAZE_PM_G1', ETcVnDiffusivityTypeKAZE.TCVN_DT1_KAZE_PM_G1);
AddLocalEnumeration('TCVN_DT1_KAZE_PM_G2', ETcVnDiffusivityTypeKAZE.TCVN_DT1_KAZE_PM_G2);
AddLocalEnumeration('TCVN_DT1_KAZE_WEICKERT', ETcVnDiffusivityTypeKAZE.TCVN_DT1_KAZE_WEICKERT);
AddLocalEnumeration('TCVN_DT1_KAZE_CHARBONNIER', ETcVnDiffusivityTypeKAZE.TCVN_DT1_KAZE_CHARBONNIER);
END_METHOD

METHOD PRIVATE AddLocalEnumeration
VAR_INPUT
	Enumeration : T_MAXSTRING;
	Value : ETcVnDiffusivityTypeKAZE;
END_VAR
AddEnumeration(Enumeration, Value);
END_METHOD

METHOD IsEnumeratorValueEqual : BOOL
VAR_INPUT
	Enumerator : I_KeyValueForwardEnumerator;
END_VAR
VAR
	storedValue : ETcVnDiffusivityTypeKAZE;
END_VAR
IF NOT Enumerator.TryGet(storedValue) THEN
	RETURN;
END_IF

IsEnumeratorValueEqual := storedValue = activeData;
END_METHOD

METHOD PUBLIC Clone : I_Datatype
VAR
    pClone : POINTER TO _ETcVnDiffusivityTypeKAZE;
END_VAR
pClone := __NEW(_ETcVnDiffusivityTypeKAZE(InitialValue := Value));
Clone := pClone^;
END_METHOD

PROPERTY PUBLIC Identifier : T_MAXSTRING
GET
Identifier := 'ETcVnDiffusivityTypeKAZE';
END_GET
END_PROPERTY

METHOD PUBLIC MakeReferenceTo
VAR_INPUT
	ReferenceTarget : REFERENCE TO ETcVnDiffusivityTypeKAZE;
END_VAR
activeData REF= ReferenceTarget;
SetBaseDatatypeReference();
END_METHOD

METHOD TryMakeReferenceTo : BOOL
VAR_INPUT
	Target : I_Datatype;
END_VAR
VAR
	pTargetData : POINTER TO ETcVnDiffusivityTypeKAZE;
END_VAR
IF NOT IsEquivalentTo(Target) THEN
	RETURN;
END_IF

pTargetData := Target.Address;
activeData REF= pTargetData^;
SetBaseDatatypeReference();
TryMakeReferenceTo := TRUE;
END_METHOD

PROPERTY PUBLIC Value : ETcVnDiffusivityTypeKAZE
GET
Value := activeData;
END_GET
SET
activeData := Value;
END_SET
END_PROPERTY

END_FUNCTION_BLOCK

// Datatypes/Enums/_ETcVnDistanceTransformationLabel
{attribute 'linkalways'} 
{attribute 'no_explicit_call' := 'This FB is a CLASS and must be accessed using methods or properties'}
{attribute 'enable_dynamic_creation'}
FUNCTION_BLOCK _ETcVnDistanceTransformationLabel EXTENDS EnumDatatypeBase
VAR
	localData : ETcVnDistanceTransformationLabel;
	activeData : REFERENCE TO ETcVnDistanceTransformationLabel;
	enumBaseDatatype : _DINT(localData);
END_VAR

METHOD PROTECTED SetBaseDatatypeReference
VAR_INPUT
END_VAR
enumBaseDatatype.MakeReferenceTo(activeData);
END_METHOD

PROPERTY PUBLIC Address : PVOID
GET
Address := ADR(activeData);
END_GET
END_PROPERTY

METHOD PUBLIC ClearReference
VAR_INPUT
END_VAR
activeData REF= localData;
SetBaseDatatypeReference();
END_METHOD

PROPERTY PUBLIC Size : UDINT
GET
Size := SIZEOF(activeData);
END_GET
END_PROPERTY

METHOD FB_init : BOOL
VAR_INPUT
	bInitRetains : BOOL; // if TRUE, the retain variables are initialized (warm start / cold start)
	bInCopyCode : BOOL;  // if TRUE, the instance afterwards gets moved into the copy code (online change)
	InitialValue : ETcVnDistanceTransformationLabel;
END_VAR
localData := InitialValue;
AddBaseDatatype(enumBaseDatatype);
ClearReference();

AddLocalEnumeration('TCVN_DTL_CCOMP', ETcVnDistanceTransformationLabel.TCVN_DTL_CCOMP);
AddLocalEnumeration('TCVN_DTL_PIXEL', ETcVnDistanceTransformationLabel.TCVN_DTL_PIXEL);
END_METHOD

METHOD PRIVATE AddLocalEnumeration
VAR_INPUT
	Enumeration : T_MAXSTRING;
	Value : ETcVnDistanceTransformationLabel;
END_VAR
AddEnumeration(Enumeration, Value);
END_METHOD

METHOD IsEnumeratorValueEqual : BOOL
VAR_INPUT
	Enumerator : I_KeyValueForwardEnumerator;
END_VAR
VAR
	storedValue : ETcVnDistanceTransformationLabel;
END_VAR
IF NOT Enumerator.TryGet(storedValue) THEN
	RETURN;
END_IF

IsEnumeratorValueEqual := storedValue = activeData;
END_METHOD

METHOD PUBLIC Clone : I_Datatype
VAR
    pClone : POINTER TO _ETcVnDistanceTransformationLabel;
END_VAR
pClone := __NEW(_ETcVnDistanceTransformationLabel(InitialValue := Value));
Clone := pClone^;
END_METHOD

PROPERTY PUBLIC Identifier : T_MAXSTRING
GET
Identifier := 'ETcVnDistanceTransformationLabel';
END_GET
END_PROPERTY

METHOD PUBLIC MakeReferenceTo
VAR_INPUT
	ReferenceTarget : REFERENCE TO ETcVnDistanceTransformationLabel;
END_VAR
activeData REF= ReferenceTarget;
SetBaseDatatypeReference();
END_METHOD

METHOD TryMakeReferenceTo : BOOL
VAR_INPUT
	Target : I_Datatype;
END_VAR
VAR
	pTargetData : POINTER TO ETcVnDistanceTransformationLabel;
END_VAR
IF NOT IsEquivalentTo(Target) THEN
	RETURN;
END_IF

pTargetData := Target.Address;
activeData REF= pTargetData^;
SetBaseDatatypeReference();
TryMakeReferenceTo := TRUE;
END_METHOD

PROPERTY PUBLIC Value : ETcVnDistanceTransformationLabel
GET
Value := activeData;
END_GET
SET
activeData := Value;
END_SET
END_PROPERTY

END_FUNCTION_BLOCK

// Datatypes/Enums/_ETcVnDistanceTransformationMask
{attribute 'linkalways'} 
{attribute 'no_explicit_call' := 'This FB is a CLASS and must be accessed using methods or properties'}
{attribute 'enable_dynamic_creation'}
FUNCTION_BLOCK _ETcVnDistanceTransformationMask EXTENDS EnumDatatypeBase
VAR
	localData : ETcVnDistanceTransformationMask;
	activeData : REFERENCE TO ETcVnDistanceTransformationMask;
	enumBaseDatatype : _DINT(localData);
END_VAR

METHOD PROTECTED SetBaseDatatypeReference
VAR_INPUT
END_VAR
enumBaseDatatype.MakeReferenceTo(activeData);
END_METHOD

PROPERTY PUBLIC Address : PVOID
GET
Address := ADR(activeData);
END_GET
END_PROPERTY

METHOD PUBLIC ClearReference
VAR_INPUT
END_VAR
activeData REF= localData;
SetBaseDatatypeReference();
END_METHOD

PROPERTY PUBLIC Size : UDINT
GET
Size := SIZEOF(activeData);
END_GET
END_PROPERTY

METHOD FB_init : BOOL
VAR_INPUT
	bInitRetains : BOOL; // if TRUE, the retain variables are initialized (warm start / cold start)
	bInCopyCode : BOOL;  // if TRUE, the instance afterwards gets moved into the copy code (online change)
	InitialValue : ETcVnDistanceTransformationMask;
END_VAR
localData := InitialValue;
AddBaseDatatype(enumBaseDatatype);
ClearReference();

AddLocalEnumeration('TCVN_DTM_PRECISE', ETcVnDistanceTransformationMask.TCVN_DTM_PRECISE);
AddLocalEnumeration('TCVN_DTM_3', ETcVnDistanceTransformationMask.TCVN_DTM_3);
AddLocalEnumeration('TCVN_DTM_5', ETcVnDistanceTransformationMask.TCVN_DTM_5);
END_METHOD

METHOD PRIVATE AddLocalEnumeration
VAR_INPUT
	Enumeration : T_MAXSTRING;
	Value : ETcVnDistanceTransformationMask;
END_VAR
AddEnumeration(Enumeration, Value);
END_METHOD

METHOD IsEnumeratorValueEqual : BOOL
VAR_INPUT
	Enumerator : I_KeyValueForwardEnumerator;
END_VAR
VAR
	storedValue : ETcVnDistanceTransformationMask;
END_VAR
IF NOT Enumerator.TryGet(storedValue) THEN
	RETURN;
END_IF

IsEnumeratorValueEqual := storedValue = activeData;
END_METHOD

METHOD PUBLIC Clone : I_Datatype
VAR
    pClone : POINTER TO _ETcVnDistanceTransformationMask;
END_VAR
pClone := __NEW(_ETcVnDistanceTransformationMask(InitialValue := Value));
Clone := pClone^;
END_METHOD

PROPERTY PUBLIC Identifier : T_MAXSTRING
GET
Identifier := 'ETcVnDistanceTransformationMask';
END_GET
END_PROPERTY

METHOD PUBLIC MakeReferenceTo
VAR_INPUT
	ReferenceTarget : REFERENCE TO ETcVnDistanceTransformationMask;
END_VAR
activeData REF= ReferenceTarget;
SetBaseDatatypeReference();
END_METHOD

METHOD TryMakeReferenceTo : BOOL
VAR_INPUT
	Target : I_Datatype;
END_VAR
VAR
	pTargetData : POINTER TO ETcVnDistanceTransformationMask;
END_VAR
IF NOT IsEquivalentTo(Target) THEN
	RETURN;
END_IF

pTargetData := Target.Address;
activeData REF= pTargetData^;
SetBaseDatatypeReference();
TryMakeReferenceTo := TRUE;
END_METHOD

PROPERTY PUBLIC Value : ETcVnDistanceTransformationMask
GET
Value := activeData;
END_GET
SET
activeData := Value;
END_SET
END_PROPERTY

END_FUNCTION_BLOCK

// Datatypes/Enums/_ETcVnDistanceType
{attribute 'linkalways'} 
{attribute 'no_explicit_call' := 'This FB is a CLASS and must be accessed using methods or properties'}
{attribute 'enable_dynamic_creation'}
FUNCTION_BLOCK _ETcVnDistanceType EXTENDS EnumDatatypeBase
VAR
	localData : ETcVnDistanceType;
	activeData : REFERENCE TO ETcVnDistanceType;
	enumBaseDatatype : _DINT(localData);
END_VAR

METHOD PROTECTED SetBaseDatatypeReference
VAR_INPUT
END_VAR
enumBaseDatatype.MakeReferenceTo(activeData);
END_METHOD

PROPERTY PUBLIC Address : PVOID
GET
Address := ADR(activeData);
END_GET
END_PROPERTY

METHOD PUBLIC ClearReference
VAR_INPUT
END_VAR
activeData REF= localData;
SetBaseDatatypeReference();
END_METHOD

PROPERTY PUBLIC Size : UDINT
GET
Size := SIZEOF(activeData);
END_GET
END_PROPERTY

METHOD FB_init : BOOL
VAR_INPUT
	bInitRetains : BOOL; // if TRUE, the retain variables are initialized (warm start / cold start)
	bInCopyCode : BOOL;  // if TRUE, the instance afterwards gets moved into the copy code (online change)
	InitialValue : ETcVnDistanceType;
END_VAR
localData := InitialValue;
AddBaseDatatype(enumBaseDatatype);
ClearReference();

AddLocalEnumeration('TCVN_DT_USER', ETcVnDistanceType.TCVN_DT_USER);
AddLocalEnumeration('TCVN_DT_L1', ETcVnDistanceType.TCVN_DT_L1);
AddLocalEnumeration('TCVN_DT_L2', ETcVnDistanceType.TCVN_DT_L2);
AddLocalEnumeration('TCVN_DT_C', ETcVnDistanceType.TCVN_DT_C);
AddLocalEnumeration('TCVN_DT_L12', ETcVnDistanceType.TCVN_DT_L12);
AddLocalEnumeration('TCVN_DT_FAIR', ETcVnDistanceType.TCVN_DT_FAIR);
AddLocalEnumeration('TCVN_DT_WELSCH', ETcVnDistanceType.TCVN_DT_WELSCH);
AddLocalEnumeration('TCVN_DT_HUBER', ETcVnDistanceType.TCVN_DT_HUBER);
END_METHOD

METHOD PRIVATE AddLocalEnumeration
VAR_INPUT
	Enumeration : T_MAXSTRING;
	Value : ETcVnDistanceType;
END_VAR
AddEnumeration(Enumeration, Value);
END_METHOD

METHOD IsEnumeratorValueEqual : BOOL
VAR_INPUT
	Enumerator : I_KeyValueForwardEnumerator;
END_VAR
VAR
	storedValue : ETcVnDistanceType;
END_VAR
IF NOT Enumerator.TryGet(storedValue) THEN
	RETURN;
END_IF

IsEnumeratorValueEqual := storedValue = activeData;
END_METHOD

METHOD PUBLIC Clone : I_Datatype
VAR
    pClone : POINTER TO _ETcVnDistanceType;
END_VAR
pClone := __NEW(_ETcVnDistanceType(InitialValue := Value));
Clone := pClone^;
END_METHOD

PROPERTY PUBLIC Identifier : T_MAXSTRING
GET
Identifier := 'ETcVnDistanceType';
END_GET
END_PROPERTY

METHOD PUBLIC MakeReferenceTo
VAR_INPUT
	ReferenceTarget : REFERENCE TO ETcVnDistanceType;
END_VAR
activeData REF= ReferenceTarget;
SetBaseDatatypeReference();
END_METHOD

METHOD TryMakeReferenceTo : BOOL
VAR_INPUT
	Target : I_Datatype;
END_VAR
VAR
	pTargetData : POINTER TO ETcVnDistanceType;
END_VAR
IF NOT IsEquivalentTo(Target) THEN
	RETURN;
END_IF

pTargetData := Target.Address;
activeData REF= pTargetData^;
SetBaseDatatypeReference();
TryMakeReferenceTo := TRUE;
END_METHOD

PROPERTY PUBLIC Value : ETcVnDistanceType
GET
Value := activeData;
END_GET
SET
activeData := Value;
END_SET
END_PROPERTY

METHOD PUBLIC TryDeserializeFrom : BOOL
VAR_INPUT
    Deserializer : I_Deserializer;
    Feedback : I_DeserializerFeedback;
END_VAR
VAR
    key : T_MAXSTRING;
END_VAR
// Accept the label emitted by older versions, but serialize the canonical label.
IF NOT Deserializer.TryGetString(key, Feedback) THEN
    RETURN;
END_IF

IF key = 'TCVN_DT_HUBER ' THEN
    activeData := ETcVnDistanceType.TCVN_DT_HUBER;
    TryDeserializeFrom := TRUE;
    RETURN;
END_IF

TryDeserializeFrom := SUPER^.TryDeserializeFrom(Deserializer, Feedback);
END_METHOD

END_FUNCTION_BLOCK

// Datatypes/Enums/_ETcVnDotCodeOptions
{attribute 'linkalways'}
{attribute 'no_explicit_call' := 'This FB is a CLASS and must be accessed using methods or properties'}
{attribute 'enable_dynamic_creation'}
FUNCTION_BLOCK _ETcVnDotCodeOptions EXTENDS EnumDatatypeBase
VAR
	localData : ETcVnDotCodeOptions;
	activeData : REFERENCE TO ETcVnDotCodeOptions;
	enumBaseDatatype : _ULINT(localData);
END_VAR

METHOD PROTECTED SetBaseDatatypeReference
VAR_INPUT
END_VAR
enumBaseDatatype.MakeReferenceTo(activeData);
END_METHOD

PROPERTY PUBLIC Address : PVOID
GET
Address := ADR(activeData);
END_GET
END_PROPERTY

METHOD PUBLIC ClearReference
VAR_INPUT
END_VAR
activeData REF= localData;
SetBaseDatatypeReference();
END_METHOD

PROPERTY PUBLIC Size : UDINT
GET
Size := SIZEOF(activeData);
END_GET
END_PROPERTY

METHOD FB_init : BOOL
VAR_INPUT
	bInitRetains : BOOL; // if TRUE, the retain variables are initialized (warm start / cold start)
	bInCopyCode : BOOL;  // if TRUE, the instance afterwards gets moved into the copy code (online change)
	InitialValue : ETcVnDotCodeOptions;
END_VAR
localData := InitialValue;
AddBaseDatatype(enumBaseDatatype);
ClearReference();

AddLocalEnumeration('TCVN_DCO_DEFAULT', ETcVnDotCodeOptions.TCVN_DCO_DEFAULT);
AddLocalEnumeration('TCVN_DCO_BINARY_INPUT', ETcVnDotCodeOptions.TCVN_DCO_BINARY_INPUT);
AddLocalEnumeration('TCVN_DCO_DETECTBLOBS', ETcVnDotCodeOptions.TCVN_DCO_DETECTBLOBS);
AddLocalEnumeration('TCVN_DCO_FILTERCONTOURS', ETcVnDotCodeOptions.TCVN_DCO_FILTERCONTOURS);
AddLocalEnumeration('TCVN_DCO_REGULAR_COLOR', ETcVnDotCodeOptions.TCVN_DCO_REGULAR_COLOR);
AddLocalEnumeration('TCVN_DCO_INVERTED_COLOR', ETcVnDotCodeOptions.TCVN_DCO_INVERTED_COLOR);
END_METHOD

METHOD PRIVATE AddLocalEnumeration
VAR_INPUT
	Enumeration : T_MAXSTRING;
	Value : ETcVnDotCodeOptions;
END_VAR
AddEnumeration(Enumeration, Value);
END_METHOD

METHOD IsEnumeratorValueEqual : BOOL
VAR_INPUT
	Enumerator : I_KeyValueForwardEnumerator;
END_VAR
VAR
	storedValue : ETcVnDotCodeOptions;
END_VAR
IF NOT Enumerator.TryGet(storedValue) THEN
	RETURN;
END_IF

IsEnumeratorValueEqual := storedValue = activeData;
END_METHOD

METHOD PUBLIC Clone : I_Datatype
VAR
    pClone : POINTER TO _ETcVnDotCodeOptions;
END_VAR
pClone := __NEW(_ETcVnDotCodeOptions(InitialValue := Value));
IF pClone = 0 THEN
    RETURN;
END_IF
Clone := pClone^;
END_METHOD

PROPERTY PUBLIC Identifier : T_MAXSTRING
GET
Identifier := 'ETcVnDotCodeOptions';
END_GET
END_PROPERTY

METHOD PUBLIC MakeReferenceTo
VAR_INPUT
	ReferenceTarget : REFERENCE TO ETcVnDotCodeOptions;
END_VAR
activeData REF= ReferenceTarget;
SetBaseDatatypeReference();
END_METHOD

METHOD TryMakeReferenceTo : BOOL
VAR_INPUT
	Target : I_Datatype;
END_VAR
VAR
	pTargetData : POINTER TO ETcVnDotCodeOptions;
END_VAR
IF NOT IsEquivalentTo(Target) THEN
	RETURN;
END_IF

pTargetData := Target.Address;
activeData REF= pTargetData^;
SetBaseDatatypeReference();
TryMakeReferenceTo := TRUE;
END_METHOD

PROPERTY PUBLIC Value : ETcVnDotCodeOptions
GET
Value := activeData;
END_GET
SET
activeData := Value;
END_SET
END_PROPERTY

END_FUNCTION_BLOCK

// Datatypes/Enums/_ETcVnDrawMatchesFlags
{attribute 'linkalways'} 
{attribute 'no_explicit_call' := 'This FB is a CLASS and must be accessed using methods or properties'}
{attribute 'enable_dynamic_creation'}
FUNCTION_BLOCK _ETcVnDrawMatchesFlags EXTENDS EnumDatatypeBase
VAR
	localData : ETcVnDrawMatchesFlags;
	activeData : REFERENCE TO ETcVnDrawMatchesFlags;
	enumBaseDatatype : _DINT(localData);
END_VAR

METHOD PROTECTED SetBaseDatatypeReference
VAR_INPUT
END_VAR
enumBaseDatatype.MakeReferenceTo(activeData);
END_METHOD

PROPERTY PUBLIC Address : PVOID
GET
Address := ADR(activeData);
END_GET
END_PROPERTY

METHOD PUBLIC ClearReference
VAR_INPUT
END_VAR
activeData REF= localData;
SetBaseDatatypeReference();
END_METHOD

PROPERTY PUBLIC Size : UDINT
GET
Size := SIZEOF(activeData);
END_GET
END_PROPERTY

METHOD FB_init : BOOL
VAR_INPUT
	bInitRetains : BOOL; // if TRUE, the retain variables are initialized (warm start / cold start)
	bInCopyCode : BOOL;  // if TRUE, the instance afterwards gets moved into the copy code (online change)
	InitialValue : ETcVnDrawMatchesFlags;
END_VAR
localData := InitialValue;
AddBaseDatatype(enumBaseDatatype);
ClearReference();

AddLocalEnumeration('TCVN_DMF_DEFAULT', ETcVnDrawMatchesFlags.TCVN_DMF_DEFAULT);
AddLocalEnumeration('TCVN_DMF_OVERDRAW', ETcVnDrawMatchesFlags.TCVN_DMF_OVERDRAW);
AddLocalEnumeration('TCVN_DMF_SKIPSINGLE', ETcVnDrawMatchesFlags.TCVN_DMF_SKIPSINGLE);
AddLocalEnumeration('TCVN_DMF_OVERDRAW_SKIPSINGLE', ETcVnDrawMatchesFlags.TCVN_DMF_OVERDRAW_SKIPSINGLE);
AddLocalEnumeration('TCVN_DMF_RICHKEYPOINT', ETcVnDrawMatchesFlags.TCVN_DMF_RICHKEYPOINT);
AddLocalEnumeration('TCVN_DMF_OVERDRAW_RICHKEYPOINT', ETcVnDrawMatchesFlags.TCVN_DMF_OVERDRAW_RICHKEYPOINT);
AddLocalEnumeration('TCVN_DMF_SKIPSINGLE_RICHKEYPOINT', ETcVnDrawMatchesFlags.TCVN_DMF_SKIPSINGLE_RICHKEYPOINT);
AddLocalEnumeration('TCVN_DMF_OVERDRAW_SKIPSINGLE_RICHKEYPOINT', ETcVnDrawMatchesFlags.TCVN_DMF_OVERDRAW_SKIPSINGLE_RICHKEYPOINT);
END_METHOD

METHOD PRIVATE AddLocalEnumeration
VAR_INPUT
	Enumeration : T_MAXSTRING;
	Value : ETcVnDrawMatchesFlags;
END_VAR
AddEnumeration(Enumeration, Value);
END_METHOD

METHOD IsEnumeratorValueEqual : BOOL
VAR_INPUT
	Enumerator : I_KeyValueForwardEnumerator;
END_VAR
VAR
	storedValue : ETcVnDrawMatchesFlags;
END_VAR
IF NOT Enumerator.TryGet(storedValue) THEN
	RETURN;
END_IF

IsEnumeratorValueEqual := storedValue = activeData;
END_METHOD

METHOD PUBLIC Clone : I_Datatype
VAR
    pClone : POINTER TO _ETcVnDrawMatchesFlags;
END_VAR
pClone := __NEW(_ETcVnDrawMatchesFlags(InitialValue := Value));
Clone := pClone^;
END_METHOD

PROPERTY PUBLIC Identifier : T_MAXSTRING
GET
Identifier := 'ETcVnDrawMatchesFlags';
END_GET
END_PROPERTY

METHOD PUBLIC MakeReferenceTo
VAR_INPUT
	ReferenceTarget : REFERENCE TO ETcVnDrawMatchesFlags;
END_VAR
activeData REF= ReferenceTarget;
SetBaseDatatypeReference();
END_METHOD

METHOD TryMakeReferenceTo : BOOL
VAR_INPUT
	Target : I_Datatype;
END_VAR
VAR
	pTargetData : POINTER TO ETcVnDrawMatchesFlags;
END_VAR
IF NOT IsEquivalentTo(Target) THEN
	RETURN;
END_IF

pTargetData := Target.Address;
activeData REF= pTargetData^;
SetBaseDatatypeReference();
TryMakeReferenceTo := TRUE;
END_METHOD

PROPERTY PUBLIC Value : ETcVnDrawMatchesFlags
GET
Value := activeData;
END_GET
SET
activeData := Value;
END_SET
END_PROPERTY

END_FUNCTION_BLOCK

// Datatypes/Enums/_ETcVnDrawShape
{attribute 'linkalways'} 
{attribute 'no_explicit_call' := 'This FB is a CLASS and must be accessed using methods or properties'}
{attribute 'enable_dynamic_creation'}
FUNCTION_BLOCK _ETcVnDrawShape EXTENDS EnumDatatypeBase
VAR
	localData : ETcVnDrawShape;
	activeData : REFERENCE TO ETcVnDrawShape;
	enumBaseDatatype : _DINT(localData);
END_VAR

METHOD PROTECTED SetBaseDatatypeReference
VAR_INPUT
END_VAR
enumBaseDatatype.MakeReferenceTo(activeData);
END_METHOD

PROPERTY PUBLIC Address : PVOID
GET
Address := ADR(activeData);
END_GET
END_PROPERTY

METHOD PUBLIC ClearReference
VAR_INPUT
END_VAR
activeData REF= localData;
SetBaseDatatypeReference();
END_METHOD

PROPERTY PUBLIC Size : UDINT
GET
Size := SIZEOF(activeData);
END_GET
END_PROPERTY

METHOD FB_init : BOOL
VAR_INPUT
	bInitRetains : BOOL; // if TRUE, the retain variables are initialized (warm start / cold start)
	bInCopyCode : BOOL;  // if TRUE, the instance afterwards gets moved into the copy code (online change)
	InitialValue : ETcVnDrawShape;
END_VAR
localData := InitialValue;
AddBaseDatatype(enumBaseDatatype);
ClearReference();

AddLocalEnumeration('TCVN_DS_RANDOM', ETcVnDrawShape.TCVN_DS_RANDOM);
AddLocalEnumeration('TCVN_DS_CIRCLE', ETcVnDrawShape.TCVN_DS_CIRCLE);
AddLocalEnumeration('TCVN_DS_SQUARE', ETcVnDrawShape.TCVN_DS_SQUARE);
AddLocalEnumeration('TCVN_DS_PLUS', ETcVnDrawShape.TCVN_DS_PLUS);
AddLocalEnumeration('TCVN_DS_X', ETcVnDrawShape.TCVN_DS_X);
AddLocalEnumeration('TCVN_DS_DIAMOND', ETcVnDrawShape.TCVN_DS_DIAMOND);
AddLocalEnumeration('TCVN_DS_MAX', ETcVnDrawShape.TCVN_DS_MAX);
END_METHOD

METHOD PRIVATE AddLocalEnumeration
VAR_INPUT
	Enumeration : T_MAXSTRING;
	Value : ETcVnDrawShape;
END_VAR
AddEnumeration(Enumeration, Value);
END_METHOD

METHOD IsEnumeratorValueEqual : BOOL
VAR_INPUT
	Enumerator : I_KeyValueForwardEnumerator;
END_VAR
VAR
	storedValue : ETcVnDrawShape;
END_VAR
IF NOT Enumerator.TryGet(storedValue) THEN
	RETURN;
END_IF

IsEnumeratorValueEqual := storedValue = activeData;
END_METHOD

METHOD PUBLIC Clone : I_Datatype
VAR
    pClone : POINTER TO _ETcVnDrawShape;
END_VAR
pClone := __NEW(_ETcVnDrawShape(InitialValue := Value));
Clone := pClone^;
END_METHOD

PROPERTY PUBLIC Identifier : T_MAXSTRING
GET
Identifier := 'ETcVnDrawShape';
END_GET
END_PROPERTY

METHOD PUBLIC MakeReferenceTo
VAR_INPUT
	ReferenceTarget : REFERENCE TO ETcVnDrawShape;
END_VAR
activeData REF= ReferenceTarget;
SetBaseDatatypeReference();
END_METHOD

METHOD TryMakeReferenceTo : BOOL
VAR_INPUT
	Target : I_Datatype;
END_VAR
VAR
	pTargetData : POINTER TO ETcVnDrawShape;
END_VAR
IF NOT IsEquivalentTo(Target) THEN
	RETURN;
END_IF

pTargetData := Target.Address;
activeData REF= pTargetData^;
SetBaseDatatypeReference();
TryMakeReferenceTo := TRUE;
END_METHOD

PROPERTY PUBLIC Value : ETcVnDrawShape
GET
Value := activeData;
END_GET
SET
activeData := Value;
END_SET
END_PROPERTY

END_FUNCTION_BLOCK

// Datatypes/Enums/_ETcVnEdgeDetectionAlgorithm
{attribute 'linkalways'} 
{attribute 'no_explicit_call' := 'This FB is a CLASS and must be accessed using methods or properties'}
{attribute 'enable_dynamic_creation'}
FUNCTION_BLOCK _ETcVnEdgeDetectionAlgorithm EXTENDS EnumDatatypeBase
VAR
	localData : ETcVnEdgeDetectionAlgorithm;
	activeData : REFERENCE TO ETcVnEdgeDetectionAlgorithm;
	enumBaseDatatype : _DINT(localData);
END_VAR

METHOD PROTECTED SetBaseDatatypeReference
VAR_INPUT
END_VAR
enumBaseDatatype.MakeReferenceTo(activeData);
END_METHOD

PROPERTY PUBLIC Address : PVOID
GET
Address := ADR(activeData);
END_GET
END_PROPERTY

METHOD PUBLIC ClearReference
VAR_INPUT
END_VAR
activeData REF= localData;
SetBaseDatatypeReference();
END_METHOD

PROPERTY PUBLIC Size : UDINT
GET
Size := SIZEOF(activeData);
END_GET
END_PROPERTY

METHOD FB_init : BOOL
VAR_INPUT
	bInitRetains : BOOL; // if TRUE, the retain variables are initialized (warm start / cold start)
	bInCopyCode : BOOL;  // if TRUE, the instance afterwards gets moved into the copy code (online change)
	InitialValue : ETcVnEdgeDetectionAlgorithm;
END_VAR
localData := InitialValue;
AddBaseDatatype(enumBaseDatatype);
ClearReference();

AddLocalEnumeration('TCVN_EDA_INTERPOLATION', ETcVnEdgeDetectionAlgorithm.TCVN_EDA_INTERPOLATION);
AddLocalEnumeration('TCVN_EDA_APPROX_ERF', ETcVnEdgeDetectionAlgorithm.TCVN_EDA_APPROX_ERF);
AddLocalEnumeration('TCVN_EDA_APPROX_GAUSSIAN', ETcVnEdgeDetectionAlgorithm.TCVN_EDA_APPROX_GAUSSIAN);
END_METHOD

METHOD PRIVATE AddLocalEnumeration
VAR_INPUT
	Enumeration : T_MAXSTRING;
	Value : ETcVnEdgeDetectionAlgorithm;
END_VAR
AddEnumeration(Enumeration, Value);
END_METHOD

METHOD IsEnumeratorValueEqual : BOOL
VAR_INPUT
	Enumerator : I_KeyValueForwardEnumerator;
END_VAR
VAR
	storedValue : ETcVnEdgeDetectionAlgorithm;
END_VAR
IF NOT Enumerator.TryGet(storedValue) THEN
	RETURN;
END_IF

IsEnumeratorValueEqual := storedValue = activeData;
END_METHOD

METHOD PUBLIC Clone : I_Datatype
VAR
    pClone : POINTER TO _ETcVnEdgeDetectionAlgorithm;
END_VAR
pClone := __NEW(_ETcVnEdgeDetectionAlgorithm(InitialValue := Value));
Clone := pClone^;
END_METHOD

PROPERTY PUBLIC Identifier : T_MAXSTRING
GET
Identifier := 'ETcVnEdgeDetectionAlgorithm';
END_GET
END_PROPERTY

METHOD PUBLIC MakeReferenceTo
VAR_INPUT
	ReferenceTarget : REFERENCE TO ETcVnEdgeDetectionAlgorithm;
END_VAR
activeData REF= ReferenceTarget;
SetBaseDatatypeReference();
END_METHOD

METHOD TryMakeReferenceTo : BOOL
VAR_INPUT
	Target : I_Datatype;
END_VAR
VAR
	pTargetData : POINTER TO ETcVnEdgeDetectionAlgorithm;
END_VAR
IF NOT IsEquivalentTo(Target) THEN
	RETURN;
END_IF

pTargetData := Target.Address;
activeData REF= pTargetData^;
SetBaseDatatypeReference();
TryMakeReferenceTo := TRUE;
END_METHOD

PROPERTY PUBLIC Value : ETcVnEdgeDetectionAlgorithm
GET
Value := activeData;
END_GET
SET
activeData := Value;
END_SET
END_PROPERTY

END_FUNCTION_BLOCK

// Datatypes/Enums/_ETcVnEdgeDirection
{attribute 'linkalways'} 
{attribute 'no_explicit_call' := 'This FB is a CLASS and must be accessed using methods or properties'}
{attribute 'enable_dynamic_creation'}
FUNCTION_BLOCK _ETcVnEdgeDirection EXTENDS EnumDatatypeBase
VAR
	localData : ETcVnEdgeDirection;
	activeData : REFERENCE TO ETcVnEdgeDirection;
	enumBaseDatatype : _DINT(localData);
END_VAR

METHOD PROTECTED SetBaseDatatypeReference
VAR_INPUT
END_VAR
enumBaseDatatype.MakeReferenceTo(activeData);
END_METHOD

PROPERTY PUBLIC Address : PVOID
GET
Address := ADR(activeData);
END_GET
END_PROPERTY

METHOD PUBLIC ClearReference
VAR_INPUT
END_VAR
activeData REF= localData;
SetBaseDatatypeReference();
END_METHOD

PROPERTY PUBLIC Size : UDINT
GET
Size := SIZEOF(activeData);
END_GET
END_PROPERTY

METHOD FB_init : BOOL
VAR_INPUT
	bInitRetains : BOOL; // if TRUE, the retain variables are initialized (warm start / cold start)
	bInCopyCode : BOOL;  // if TRUE, the instance afterwards gets moved into the copy code (online change)
	InitialValue : ETcVnEdgeDirection;
END_VAR
localData := InitialValue;
AddBaseDatatype(enumBaseDatatype);
ClearReference();

AddLocalEnumeration('TCVN_ED_DARK_TO_LIGHT', ETcVnEdgeDirection.TCVN_ED_DARK_TO_LIGHT);
AddLocalEnumeration('TCVN_ED_LIGHT_TO_DARK', ETcVnEdgeDirection.TCVN_ED_LIGHT_TO_DARK);
END_METHOD

METHOD PRIVATE AddLocalEnumeration
VAR_INPUT
	Enumeration : T_MAXSTRING;
	Value : ETcVnEdgeDirection;
END_VAR
AddEnumeration(Enumeration, Value);
END_METHOD

METHOD IsEnumeratorValueEqual : BOOL
VAR_INPUT
	Enumerator : I_KeyValueForwardEnumerator;
END_VAR
VAR
	storedValue : ETcVnEdgeDirection;
END_VAR
IF NOT Enumerator.TryGet(storedValue) THEN
	RETURN;
END_IF

IsEnumeratorValueEqual := storedValue = activeData;
END_METHOD

METHOD PUBLIC Clone : I_Datatype
VAR
    pClone : POINTER TO _ETcVnEdgeDirection;
END_VAR
pClone := __NEW(_ETcVnEdgeDirection(InitialValue := Value));
Clone := pClone^;
END_METHOD

PROPERTY PUBLIC Identifier : T_MAXSTRING
GET
Identifier := 'ETcVnEdgeDirection';
END_GET
END_PROPERTY

METHOD PUBLIC MakeReferenceTo
VAR_INPUT
	ReferenceTarget : REFERENCE TO ETcVnEdgeDirection;
END_VAR
activeData REF= ReferenceTarget;
SetBaseDatatypeReference();
END_METHOD

METHOD TryMakeReferenceTo : BOOL
VAR_INPUT
	Target : I_Datatype;
END_VAR
VAR
	pTargetData : POINTER TO ETcVnEdgeDirection;
END_VAR
IF NOT IsEquivalentTo(Target) THEN
	RETURN;
END_IF

pTargetData := Target.Address;
activeData REF= pTargetData^;
SetBaseDatatypeReference();
TryMakeReferenceTo := TRUE;
END_METHOD

PROPERTY PUBLIC Value : ETcVnEdgeDirection
GET
Value := activeData;
END_GET
SET
activeData := Value;
END_SET
END_PROPERTY

END_FUNCTION_BLOCK

// Datatypes/Enums/_ETcVnEdgeSelection
{attribute 'linkalways'}
{attribute 'no_explicit_call' := 'This FB is a CLASS and must be accessed using methods or properties'}
{attribute 'enable_dynamic_creation'}
FUNCTION_BLOCK _ETcVnEdgeSelection EXTENDS EnumDatatypeBase
VAR
	localData : ETcVnEdgeSelection;
	activeData : REFERENCE TO ETcVnEdgeSelection;
	enumBaseDatatype : _DINT(localData);
END_VAR

METHOD PROTECTED SetBaseDatatypeReference
VAR_INPUT
END_VAR
enumBaseDatatype.MakeReferenceTo(activeData);
END_METHOD

PROPERTY PUBLIC Address : PVOID
GET
Address := ADR(activeData);
END_GET
END_PROPERTY

METHOD PUBLIC ClearReference
VAR_INPUT
END_VAR
activeData REF= localData;
SetBaseDatatypeReference();
END_METHOD

PROPERTY PUBLIC Size : UDINT
GET
Size := SIZEOF(activeData);
END_GET
END_PROPERTY

METHOD FB_init : BOOL
VAR_INPUT
	bInitRetains : BOOL; // if TRUE, the retain variables are initialized (warm start / cold start)
	bInCopyCode : BOOL;  // if TRUE, the instance afterwards gets moved into the copy code (online change)
	InitialValue : ETcVnEdgeSelection;
END_VAR
localData := InitialValue;
AddBaseDatatype(enumBaseDatatype);
ClearReference();

